C09031=1032.657,-130.353,-79.572,167.440,40.256,157.483
C09032=1032.659,-130.603,-79.558,167.438,40.252,157.482
C09033=1032.660,-130.853,-79.542,167.436,40.248,157.482
C09034=1032.663,-131.102,-79.526,167.435,40.244,157.481
C09035=1032.666,-131.352,-79.509,167.433,40.239,157.480
C09036=1032.671,-131.603,-79.492,167.432,40.234,157.479
C09037=1032.675,-131.852,-79.475,167.431,40.228,157.478
C09038=1032.681,-132.102,-79.456,167.430,40.222,157.477
C09039=1032.354,-132.127,-79.747,167.381,40.451,157.513
C09040=1032.348,-131.877,-79.766,167.383,40.457,157.514
C09041=1032.344,-131.627,-79.784,167.384,40.463,157.515
C09042=1032.340,-131.377,-79.801,167.385,40.468,157.516
C09043=1032.337,-131.127,-79.818,167.386,40.473,157.517
C09044=1032.333,-130.877,-79.834,167.388,40.478,157.518
C09045=1032.331,-130.627,-79.849,167.390,40.482,157.519
C09046=1032.330,-130.377,-79.864,167.391,40.485,157.519
C09047=1032.330,-130.127,-79.879,167.393,40.488,157.520
C09048=1032.330,-129.877,-79.892,167.395,40.490,157.520
C09049=1032.331,-129.628,-79.905,167.397,40.492,157.521
C09050=1032.331,-129.377,-79.918,167.400,40.494,157.521
C09051=1032.334,-129.128,-79.930,167.402,40.495,157.521
C09052=1032.336,-128.878,-79.941,167.404,40.496,157.522
C09053=1032.339,-128.629,-79.952,167.406,40.495,157.522
C09054=1032.343,-128.379,-79.962,167.409,40.495,157.522
C09055=1032.348,-128.129,-79.971,167.411,40.495,157.522
C09056=1032.353,-127.880,-79.981,167.414,40.493,157.522
C09057=1032.359,-127.629,-79.990,167.417,40.492,157.522
C09058=1032.364,-127.380,-79.998,167.419,40.490,157.521
C09059=1032.371,-127.131,-80.007,167.422,40.488,157.521
C09060=1032.376,-126.881,-80.015,167.425,40.487,157.521
C09061=1032.382,-126.631,-80.023,167.428,40.485,157.521
C09062=1032.388,-126.381,-80.032,167.430,40.483,157.521
C09063=1032.395,-126.132,-80.041,167.434,40.482,157.521
C09064=1032.400,-125.882,-80.049,167.437,40.480,157.520
C09065=1032.406,-125.632,-80.058,167.440,40.478,157.520
C09066=1032.412,-125.382,-80.066,167.442,40.477,157.520
C09067=1032.418,-125.132,-80.075,167.445,40.475,157.520
C09068=1032.423,-124.883,-80.084,167.448,40.473,157.520
C09069=1032.430,-124.633,-80.092,167.451,40.472,157.520
C09070=1032.435,-124.383,-80.101,167.453,40.470,157.520
C09071=1032.441,-124.133,-80.110,167.456,40.469,157.520
C09072=1032.447,-123.884,-80.118,167.459,40.467,157.519
C09073=1032.453,-123.633,-80.127,167.462,40.466,157.519
C09074=1032.458,-123.384,-80.136,167.465,40.464,157.519
C09075=1032.465,-123.134,-80.145,167.467,40.462,157.519
C09076=1032.471,-122.884,-80.153,167.470,40.461,157.519
C09077=1032.477,-122.635,-80.163,167.473,40.459,157.519
C09078=1032.482,-122.385,-80.171,167.476,40.457,157.518
C09079=1032.488,-122.134,-80.180,167.479,40.456,157.518
C09080=1032.494,-121.886,-80.189,167.481,40.455,157.518
C09081=1032.500,-121.635,-80.197,167.484,40.453,157.518
C09082=1032.505,-121.386,-80.206,167.487,40.451,157.518
C09083=1032.511,-121.136,-80.216,167.490,40.450,157.518
C09084=1032.517,-120.886,-80.223,167.492,40.448,157.518
C09085=1032.524,-120.637,-80.233,167.496,40.446,157.517
C09086=1032.529,-120.387,-80.241,167.499,40.445,157.517
C09087=1032.535,-120.137,-80.251,167.502,40.444,157.517
C09088=1032.541,-119.887,-80.260,167.504,40.442,157.517
C09089=1032.547,-119.637,-80.268,167.507,40.440,157.517
C09090=1032.553,-119.387,-80.277,167.510,40.439,157.517
C09091=1032.558,-119.138,-80.286,167.513,40.437,157.517
C09092=1032.565,-118.888,-80.295,167.516,40.436,157.517
C09093=1032.570,-118.638,-80.304,167.518,40.435,157.516
C09094=1032.577,-118.389,-80.313,167.521,40.433,157.516
C09095=1032.583,-118.138,-80.322,167.524,40.431,157.516
C09096=1032.588,-117.889,-80.331,167.527,40.430,157.516
C09097=1032.594,-117.639,-80.340,167.529,40.428,157.516
C09098=1032.600,-117.389,-80.349,167.532,40.427,157.516
C09099=1032.606,-117.140,-80.358,167.535,40.425,157.516
C09100=1032.613,-116.853,-80.368,167.538,40.424,157.516
C09101=1032.620,-116.566,-80.379,167.542,40.422,157.515
C09102=1032.626,-116.280,-80.390,167.544,40.420,157.515
C09103=1032.633,-115.994,-80.400,167.548,40.418,157.515
C09104=1032.639,-115.744,-80.409,167.551,40.417,157.515
C09105=1032.645,-115.494,-80.418,167.554,40.415,157.515
C09106=1032.651,-115.245,-80.427,167.556,40.414,157.515
C09107=1032.657,-114.994,-80.436,167.559,40.413,157.515
C09108=1032.663,-114.745,-80.446,167.562,40.411,157.514
C09109=1032.669,-114.495,-80.454,167.565,40.409,157.514
C09110=1032.675,-114.245,-80.463,167.568,40.408,157.514
C09111=1032.681,-113.996,-80.473,167.570,40.407,157.514
C09112=1032.687,-113.747,-80.482,167.573,40.405,157.514
C09113=1032.693,-113.496,-80.491,167.576,40.403,157.514
C09114=1032.699,-113.246,-80.500,167.579,40.402,157.514
C09115=1032.704,-112.997,-80.510,167.582,40.401,157.514
C09116=1032.710,-112.747,-80.518,167.584,40.399,157.513
C09117=1032.716,-112.497,-80.528,167.587,40.398,157.513
C09118=1032.723,-112.247,-80.538,167.590,40.396,157.513
C09119=1032.728,-111.998,-80.547,167.593,40.395,157.513
C09120=1032.734,-111.748,-80.556,167.596,40.394,157.513
C09121=1032.740,-111.498,-80.565,167.598,40.392,157.513
C09122=1032.746,-111.248,-80.575,167.601,40.391,157.513
C09123=1032.752,-110.999,-80.584,167.604,40.390,157.513
C09124=1032.758,-110.749,-80.594,167.607,40.388,157.513
C09125=1032.764,-110.499,-80.602,167.610,40.386,157.512
C09126=1032.770,-110.249,-80.612,167.612,40.385,157.512
C09127=1032.776,-110.000,-80.621,167.615,40.384,157.512
C09128=1032.782,-109.750,-80.631,167.618,40.382,157.512
C09129=1032.787,-109.500,-80.641,167.621,40.381,157.512
C09130=1032.793,-109.250,-80.650,167.624,40.379,157.512
C09131=1032.799,-109.001,-80.660,167.626,40.378,157.512
C09132=1032.805,-108.751,-80.668,167.629,40.377,157.512
C09133=1032.811,-108.501,-80.678,167.632,40.375,157.511
C09134=1032.817,-108.251,-80.688,167.635,40.374,157.511
C09135=1032.823,-108.001,-80.697,167.638,40.373,157.511
C09136=1032.830,-107.751,-80.707,167.640,40.371,157.511
C09137=1032.835,-107.502,-80.716,167.643,40.369,157.511
C09138=1032.841,-107.253,-80.726,167.646,40.368,157.511
C09139=1032.848,-107.003,-80.735,167.649,40.367,157.511
C09140=1032.854,-106.753,-80.745,167.652,40.366,157.511
C09141=1032.860,-106.503,-80.754,167.654,40.364,157.511
C09142=1032.865,-106.253,-80.764,167.656,40.363,157.511
C09143=1032.871,-106.004,-80.774,167.659,40.362,157.510
C09144=1032.877,-105.754,-80.783,167.662,40.361,157.510
C09145=1032.883,-105.504,-80.793,167.665,40.359,157.510
C09146=1032.889,-105.255,-80.802,167.668,40.358,157.510
C09147=1032.895,-105.004,-80.812,167.670,40.356,157.510
C09148=1032.901,-104.755,-80.822,167.673,40.355,157.510
C09149=1032.907,-104.505,-80.832,167.676,40.354,157.510
C09150=1032.913,-104.256,-80.841,167.679,40.352,157.510
C09151=1032.919,-104.006,-80.850,167.682,40.351,157.510
C09152=1032.924,-103.756,-80.861,167.684,40.349,157.509
C09153=1032.931,-103.506,-80.870,167.687,40.349,157.509
C09154=1032.937,-103.256,-80.880,167.690,40.347,157.509
C09155=1032.943,-103.006,-80.889,167.693,40.346,157.509
C09156=1032.949,-102.757,-80.900,167.696,40.344,157.509
C09157=1032.955,-102.507,-80.910,167.699,40.343,157.509
C09158=1032.961,-102.257,-80.919,167.701,40.342,157.509
C09159=1032.967,-102.008,-80.929,167.704,40.341,157.509
C09160=1032.973,-101.758,-80.938,167.707,40.339,157.509
C09161=1032.978,-101.508,-80.948,167.710,40.338,157.509
C09162=1032.984,-101.259,-80.958,167.713,40.337,157.509
C09163=1032.991,-101.009,-80.968,167.715,40.336,157.508
C09164=1032.998,-100.722,-80.979,167.718,40.334,157.508
C09165=1033.004,-100.435,-80.991,167.721,40.333,157.508
C09166=1033.011,-100.148,-81.002,167.725,40.331,157.508
C09167=1033.019,-99.861,-81.013,167.728,40.330,157.508
C09168=1033.024,-99.610,-81.023,167.731,40.329,157.508
C09169=1033.031,-99.361,-81.034,167.733,40.327,157.508
C09170=1033.037,-99.111,-81.043,167.736,40.326,157.508
C09171=1033.043,-98.862,-81.053,167.739,40.324,157.507
C09172=1033.048,-98.612,-81.063,167.742,40.323,157.507
C09173=1033.055,-98.362,-81.073,167.745,40.322,157.507
C09174=1033.061,-98.113,-81.083,167.748,40.321,157.507
C09175=1033.067,-97.863,-81.092,167.750,40.319,157.507
C09176=1033.073,-97.613,-81.103,167.752,40.318,157.507
C09177=1033.079,-97.363,-81.113,167.755,40.317,157.507
C09178=1033.085,-97.113,-81.123,167.758,40.316,157.507
C09179=1033.091,-96.864,-81.133,167.761,40.315,157.507
C09180=1033.096,-96.614,-81.143,167.764,40.314,157.507
C09181=1033.103,-96.364,-81.153,167.767,40.313,157.507
C09182=1033.108,-96.115,-81.164,167.769,40.311,157.507
C09183=1033.115,-95.865,-81.173,167.772,40.310,157.506
C09184=1033.120,-95.615,-81.184,167.775,40.309,157.506
C09185=1033.126,-95.366,-81.194,167.777,40.308,157.506
C09186=1033.132,-95.116,-81.204,167.780,40.307,157.506
C09187=1033.138,-94.866,-81.215,167.783,40.306,157.506
C09188=1033.144,-94.616,-81.224,167.786,40.305,157.506
C09189=1033.150,-94.367,-81.235,167.788,40.303,157.506
C09190=1033.156,-94.117,-81.245,167.791,40.302,157.506
C09191=1033.161,-93.868,-81.256,167.794,40.301,157.506
C09192=1033.168,-93.618,-81.265,167.797,40.300,157.506
C09193=1033.173,-93.368,-81.276,167.800,40.299,157.506
C09194=1033.180,-93.118,-81.286,167.802,40.298,157.506
C09195=1033.186,-92.868,-81.297,167.805,40.297,157.506
C09196=1033.192,-92.618,-81.307,167.808,40.296,157.506
C09197=1033.198,-92.369,-81.317,167.810,40.294,157.505
C09198=1033.204,-92.119,-81.327,167.813,40.293,157.505
C09199=1033.210,-91.870,-81.338,167.816,40.292,157.505
C09200=1033.215,-91.620,-81.348,167.819,40.291,157.505
C09201=1033.222,-91.370,-81.358,167.822,40.290,157.505
C09202=1033.227,-91.121,-81.369,167.824,40.289,157.505
C09203=1033.234,-90.870,-81.379,167.826,40.288,157.505
C09204=1033.240,-90.621,-81.390,167.829,40.286,157.505
C09205=1033.246,-90.371,-81.400,167.832,40.285,157.505
C09206=1033.252,-90.122,-81.410,167.835,40.284,157.505
C09207=1033.257,-89.872,-81.421,167.838,40.283,157.505
C09208=1033.264,-89.622,-81.431,167.841,40.282,157.505
C09209=1033.269,-89.373,-81.442,167.844,40.281,157.504
C09210=1033.276,-89.123,-81.452,167.845,40.280,157.504
C09211=1033.282,-88.873,-81.463,167.848,40.279,157.504
C09212=1033.288,-88.624,-81.473,167.851,40.277,157.504
C09213=1033.294,-88.374,-81.484,167.854,40.276,157.504
C09214=1033.300,-88.124,-81.494,167.857,40.275,157.504
C09215=1033.307,-87.874,-81.505,167.860,40.274,157.504
C09216=1033.312,-87.625,-81.515,167.863,40.274,157.504
C09217=1033.319,-87.375,-81.525,167.865,40.272,157.504
C09218=1033.324,-87.125,-81.536,167.867,40.271,157.504
C09219=1033.331,-86.875,-81.547,167.870,40.270,157.504
C09220=1033.337,-86.626,-81.557,167.873,40.269,157.504
C09221=1033.343,-86.376,-81.568,167.876,40.267,157.504
C09222=1033.349,-86.127,-81.578,167.879,40.267,157.504
C09223=1033.355,-85.877,-81.589,167.882,40.266,157.503
C09224=1033.361,-85.627,-81.600,167.885,40.265,157.503
C09225=1033.367,-85.377,-81.610,167.887,40.263,157.503
C09226=1033.373,-85.128,-81.620,167.889,40.262,157.503
C09227=1033.380,-84.878,-81.631,167.892,40.261,157.503
C09228=1033.387,-84.593,-81.643,167.896,40.260,157.503
C09229=1033.394,-84.309,-81.655,167.899,40.258,157.503
C09230=1033.401,-84.023,-81.667,167.902,40.258,157.503
C09231=1033.408,-83.739,-81.679,167.904,40.256,157.503
C09232=1033.413,-83.489,-81.690,167.907,40.255,157.503
C09233=1033.420,-83.239,-81.701,167.910,40.254,157.503
C09234=1033.426,-82.990,-81.712,167.913,40.253,157.503
C09235=1033.432,-82.740,-81.722,167.916,40.251,157.503
C09236=1033.439,-82.490,-81.733,167.919,40.250,157.502
C09237=1033.444,-82.240,-81.743,167.921,40.250,157.502
C09238=1033.450,-81.991,-81.754,167.924,40.249,157.502
C09239=1033.457,-81.741,-81.765,167.926,40.248,157.502
C09240=1033.463,-81.491,-81.776,167.929,40.246,157.502
C09241=1033.469,-81.242,-81.787,167.932,40.245,157.502
C09242=1033.476,-80.992,-81.797,167.935,40.244,157.502
C09243=1033.481,-80.743,-81.808,167.938,40.243,157.502
C09244=1033.489,-80.493,-81.819,167.940,40.242,157.502
C09245=1033.494,-80.243,-81.830,167.943,40.241,157.502
C09246=1033.500,-79.994,-81.841,167.945,40.240,157.502
C09247=1033.506,-79.744,-81.852,167.948,40.239,157.502
C09248=1033.513,-79.494,-81.862,167.951,40.238,157.502
C09249=1033.519,-79.244,-81.873,167.954,40.237,157.502
C09250=1033.525,-78.995,-81.884,167.956,40.236,157.502
C09251=1033.531,-78.745,-81.895,167.959,40.235,157.502
C09252=1033.537,-78.495,-81.906,167.962,40.234,157.501
C09253=1033.543,-78.245,-81.917,167.965,40.233,157.501
C09254=1033.549,-77.996,-81.928,167.968,40.232,157.501
C09255=1033.555,-77.746,-81.939,167.969,40.231,157.501
C09256=1033.561,-77.496,-81.950,167.972,40.230,157.501
C09257=1033.568,-77.246,-81.961,167.975,40.229,157.501
C09258=1033.574,-76.998,-81.972,167.978,40.228,157.501
///RCONF 1,0,0,1,1,0,0,0,0,0,0,0,0,0,0,0,0,0,0,0,0,0,0,0
C09259=1033.579,-76.748,-81.983,167.981,40.228,157.501
C09260=1033.586,-76.498,-81.995,167.983,40.227,157.501
C09261=1033.592,-76.248,-82.005,167.986,40.226,157.501
C09262=1033.598,-75.998,-82.017,167.989,40.225,157.501
///RCONF 1,0,0,0,1,0,0,0,0,0,0,0,0,0,0,0,0,0,0,0,0,0,0,0
C09263=1033.604,-75.749,-82.028,167.992,40.224,157.501
C09264=1033.610,-75.499,-82.039,167.995,40.223,157.501
C09265=1033.616,-75.250,-82.050,167.996,40.222,157.501
C09266=1033.622,-74.999,-82.062,167.999,40.221,157.501
C09267=1033.628,-74.750,-82.072,168.002,40.219,157.501
C09268=1033.635,-74.500,-82.083,168.005,40.218,157.501
C09269=1033.641,-74.251,-82.094,168.008,40.218,157.501
C09270=1033.647,-74.002,-82.106,168.010,40.217,157.501
C09271=1033.653,-73.751,-82.117,168.013,40.216,157.501
C09272=1033.658,-73.502,-82.128,168.016,40.215,157.500
C09273=1033.665,-73.252,-82.140,168.019,40.214,157.500
///RCONF 1,0,0,0,0,0,0,0,0,0,0,0,0,0,0,0,0,0,0,0,0,0,0,0
C09274=1033.671,-73.003,-82.151,168.020,40.214,157.500
C09275=1033.677,-72.752,-82.162,168.023,40.213,157.500
C09276=1033.683,-72.504,-82.174,168.026,40.212,157.500
C09277=1033.689,-72.253,-82.186,168.028,40.212,157.500
C09278=1033.694,-72.004,-82.197,168.031,40.211,157.500
C09279=1033.701,-71.754,-82.209,168.034,40.210,157.500
C09280=1033.707,-71.505,-82.220,168.037,40.209,157.500
C09281=1033.713,-71.254,-82.231,168.039,40.208,157.500
C09282=1033.718,-71.005,-82.243,168.042,40.208,157.500
C09283=1033.725,-70.755,-82.254,168.045,40.207,157.500
C09284=1033.731,-70.506,-82.266,168.048,40.206,157.500
C09285=1033.737,-70.256,-82.277,168.050,40.205,157.500
C09286=1033.743,-70.006,-82.288,168.052,40.204,157.500
C09287=1033.749,-69.757,-82.300,168.055,40.203,157.500
C09288=1033.755,-69.507,-82.311,168.057,40.203,157.500
C09289=1033.761,-69.257,-82.323,168.060,40.202,157.500
C09290=1033.767,-69.008,-82.334,168.063,40.201,157.500
C09291=1033.774,-68.758,-82.346,168.066,40.200,157.500
C09292=1033.780,-68.476,-82.359,168.069,40.199,157.500
C09293=1033.787,-68.193,-82.372,168.072,40.198,157.500
C09294=1033.794,-67.910,-82.385,168.075,40.197,157.500
C09295=1033.801,-67.628,-82.398,168.078,40.197,157.500
C09296=1033.806,-67.377,-82.410,168.081,40.196,157.500
C09297=1033.813,-67.128,-82.422,168.083,40.195,157.500
C09298=1033.819,-66.878,-82.433,168.085,40.194,157.500
C09299=1033.825,-66.629,-82.445,168.088,40.193,157.500
C09300=1033.831,-66.380,-82.456,168.091,40.192,157.500
C09301=1033.837,-66.129,-82.468,168.093,40.192,157.500
C09302=1033.843,-65.880,-82.480,168.096,40.191,157.500
C09303=1033.849,-65.630,-82.491,168.099,40.190,157.500
C09304=1033.856,-65.381,-82.503,168.101,40.189,157.499
C09305=1033.861,-65.131,-82.514,168.104,40.188,157.499
C09306=1033.868,-64.881,-82.526,168.107,40.188,157.499
C09307=1033.874,-64.632,-82.538,168.110,40.187,157.499
C09308=1033.880,-64.382,-82.549,168.112,40.186,157.499
C09309=1033.886,-64.132,-82.562,168.115,40.185,157.499
C09310=1033.892,-63.882,-82.573,168.117,40.184,157.499
C09311=1033.898,-63.633,-82.585,168.120,40.184,157.499
C09312=1033.905,-63.384,-82.597,168.122,40.183,157.499
C09313=1033.910,-63.133,-82.608,168.125,40.182,157.499
C09314=1033.916,-62.884,-82.620,168.128,40.181,157.499
C09315=1033.923,-62.635,-82.632,168.130,40.180,157.499
C09316=1033.929,-62.384,-82.643,168.133,40.179,157.499
C09317=1033.935,-62.135,-82.656,168.136,40.179,157.499
C09318=1033.941,-61.886,-82.667,168.138,40.178,157.499
C09319=1033.948,-61.636,-82.679,168.141,40.177,157.499
C09320=1033.954,-61.386,-82.691,168.144,40.176,157.499
C09321=1033.960,-61.137,-82.703,168.146,40.175,157.499
C09322=1033.966,-60.887,-82.715,168.149,40.175,157.499
C09323=1033.973,-60.637,-82.726,168.151,40.174,157.499
C09324=1033.979,-60.387,-82.738,168.154,40.173,157.499
C09325=1033.985,-60.138,-82.750,168.156,40.172,157.499
C09326=1033.991,-59.889,-82.762,168.159,40.171,157.499
C09327=1033.998,-59.639,-82.773,168.162,40.171,157.499
C09328=1034.004,-59.389,-82.786,168.164,40.170,157.499
C09329=1034.010,-59.140,-82.797,168.167,40.169,157.499
C09330=1034.016,-58.890,-82.809,168.170,40.168,157.499
C09331=1034.023,-58.640,-82.821,168.172,40.168,157.499
C09332=1034.028,-58.390,-82.833,168.175,40.167,157.499
C09333=1034.035,-58.141,-82.845,168.178,40.166,157.499
C09334=1034.041,-57.892,-82.857,168.180,40.166,157.499
C09335=1034.047,-57.642,-82.869,168.182,40.165,157.499
C09336=1034.054,-57.392,-82.881,168.185,40.164,157.499
C09337=1034.060,-57.142,-82.893,168.188,40.163,157.499
C09338=1034.067,-56.892,-82.905,168.190,40.163,157.499
C09339=1034.073,-56.643,-82.917,168.193,40.162,157.498
C09340=1034.079,-56.394,-82.929,168.196,40.161,157.498
C09341=1034.085,-56.144,-82.941,168.198,40.160,157.498
C09342=1034.091,-55.894,-82.953,168.201,40.159,157.498
C09343=1034.098,-55.645,-82.965,168.204,40.159,157.498
C09344=1034.105,-55.395,-82.977,168.206,40.158,157.498
C09345=1034.110,-55.145,-82.989,168.209,40.157,157.498
C09346=1034.117,-54.895,-83.001,168.212,40.156,157.498
C09347=1034.123,-54.646,-83.012,168.214,40.156,157.498
C09348=1034.129,-54.396,-83.025,168.216,40.155,157.498
C09349=1034.135,-54.147,-83.037,168.219,40.154,157.498
C09350=1034.142,-53.897,-83.049,168.221,40.153,157.498
C09351=1034.148,-53.647,-83.062,168.224,40.152,157.498
C09352=1034.155,-53.398,-83.073,168.227,40.152,157.498
C09353=1034.161,-53.148,-83.085,168.229,40.151,157.498
C09354=1034.167,-52.898,-83.098,168.232,40.150,157.498
C09355=1034.174,-52.649,-83.110,168.235,40.149,157.498
C09356=1034.181,-52.368,-83.124,168.238,40.148,157.498
C09357=1034.188,-52.086,-83.137,168.241,40.147,157.498
C09358=1034.195,-51.805,-83.150,168.244,40.147,157.498
C09359=1034.202,-51.523,-83.165,168.247,40.146,157.498
C09360=1034.209,-51.274,-83.177,168.250,40.145,157.498
C09361=1034.215,-51.024,-83.189,168.251,40.144,157.498
C09362=1034.221,-50.774,-83.201,168.254,40.143,157.498
C09363=1034.228,-50.525,-83.213,168.257,40.143,157.498
C09364=1034.234,-50.275,-83.226,168.259,40.142,157.498
C09365=1034.241,-50.025,-83.238,168.262,40.141,157.498
C09366=1034.247,-49.776,-83.251,168.264,40.141,157.498
C09367=1034.253,-49.526,-83.264,168.267,40.140,157.498
C09368=1034.259,-49.276,-83.276,168.270,40.140,157.498
C09369=1034.265,-49.027,-83.288,168.272,40.139,157.498
C09370=1034.271,-48.778,-83.300,168.275,40.138,157.498
C09371=1034.277,-48.528,-83.314,168.277,40.138,157.498
C09372=1034.283,-48.279,-83.326,168.280,40.137,157.498
C09373=1034.289,-48.029,-83.338,168.282,40.136,157.498
C09374=1034.295,-47.779,-83.351,168.285,40.135,157.498
C09375=1034.302,-47.530,-83.363,168.288,40.135,157.498
C09376=1034.308,-47.280,-83.376,168.290,40.134,157.498
C09377=1034.314,-47.030,-83.388,168.293,40.134,157.498
C09378=1034.320,-46.780,-83.401,168.295,40.133,157.498
C09379=1034.327,-46.531,-83.414,168.298,40.133,157.498
C09380=1034.333,-46.282,-83.426,168.300,40.132,157.498
C09381=1034.339,-46.032,-83.439,168.302,40.132,157.498
C09382=1034.346,-45.783,-83.451,168.305,40.131,157.498
C09383=1034.352,-45.533,-83.464,168.307,40.131,157.498
C09384=1034.357,-45.283,-83.477,168.310,40.130,157.498
C09385=1034.364,-45.034,-83.490,168.313,40.129,157.498
C09386=1034.370,-44.784,-83.502,168.315,40.129,157.498
C09387=1034.376,-44.534,-83.514,168.318,40.128,157.498
C09388=1034.382,-44.285,-83.528,168.320,40.128,157.498
C09389=1034.389,-44.035,-83.540,168.323,40.127,157.498
C09390=1034.395,-43.786,-83.552,168.325,40.126,157.498
C09391=1034.401,-43.536,-83.565,168.328,40.125,157.498
C09392=1034.407,-43.286,-83.578,168.331,40.125,157.498
C09393=1034.414,-43.037,-83.590,168.333,40.124,157.498
C09394=1034.421,-42.787,-83.604,168.336,40.123,157.498
C09395=1034.426,-42.537,-83.616,168.338,40.123,157.498
C09396=1034.433,-42.288,-83.629,168.341,40.122,157.498
C09397=1034.439,-42.038,-83.641,168.343,40.122,157.498
C09398=1034.446,-41.789,-83.655,168.346,40.121,157.498
C09399=1034.451,-41.539,-83.667,168.349,40.121,157.498
C09400=1034.458,-41.290,-83.680,168.350,40.120,157.498
C09401=1034.464,-41.040,-83.692,168.354,40.120,157.498
C09402=1034.470,-40.790,-83.705,168.355,40.119,157.498
C09403=1034.476,-40.541,-83.718,168.358,40.118,157.498
C09404=1034.483,-40.290,-83.731,168.360,40.118,157.498
C09405=1034.490,-40.041,-83.744,168.363,40.117,157.498
C09406=1034.496,-39.792,-83.756,168.366,40.117,157.498
C09407=1034.502,-39.542,-83.770,168.368,40.116,157.498
C09408=1034.508,-39.292,-83.782,168.371,40.115,157.498
C09409=1034.515,-39.043,-83.795,168.373,40.115,157.498
C09410=1034.521,-38.794,-83.808,168.376,40.114,157.498
C09411=1034.528,-38.544,-83.821,168.378,40.113,157.498
C09412=1034.534,-38.294,-83.834,168.381,40.113,157.498
C09413=1034.540,-38.044,-83.847,168.383,40.112,157.498
C09414=1034.546,-37.795,-83.860,168.386,40.112,157.498
C09415=1034.552,-37.546,-83.873,168.388,40.112,157.498
C09416=1034.558,-37.296,-83.886,168.391,40.111,157.498
C09417=1034.564,-37.047,-83.899,168.393,40.111,157.498
C09418=1034.570,-36.798,-83.913,168.396,40.110,157.498
C09419=1034.577,-36.547,-83.925,168.398,40.110,157.498
C09420=1034.583,-36.267,-83.941,168.401,40.109,157.498
C09421=1034.591,-35.985,-83.955,168.404,40.108,157.498
C09422=1034.598,-35.704,-83.970,168.407,40.108,157.498
C09423=1034.604,-35.423,-83.985,168.410,40.107,157.498
C09424=1034.611,-35.174,-83.998,168.412,40.107,157.498
C09425=1034.617,-34.923,-84.011,168.415,40.106,157.498
C09426=1034.623,-34.674,-84.025,168.417,40.106,157.498
C09427=1034.629,-34.425,-84.038,168.420,40.106,157.498
C09428=1034.635,-34.175,-84.050,168.422,40.105,157.498
C09429=1034.642,-33.926,-84.064,168.425,40.104,157.498
C09430=1034.648,-33.676,-84.077,168.426,40.104,157.498
C09431=1034.655,-33.427,-84.091,168.429,40.103,157.498
C09432=1034.661,-33.177,-84.104,168.431,40.103,157.498
C09433=1034.667,-32.927,-84.116,168.434,40.102,157.498
C09434=1034.674,-32.677,-84.130,168.436,40.102,157.498
C09435=1034.680,-32.428,-84.143,168.439,40.101,157.498
C09436=1034.686,-32.179,-84.157,168.441,40.101,157.498
C09437=1034.692,-31.930,-84.170,168.444,40.101,157.498
C09438=1034.699,-31.679,-84.183,168.446,40.100,157.498
C09439=1034.705,-31.430,-84.196,168.449,40.099,157.498
C09440=1034.711,-31.181,-84.209,168.451,40.099,157.498
C09441=1034.717,-30.931,-84.223,168.454,40.098,157.498
C09442=1034.724,-30.681,-84.236,168.456,40.097,157.498
C09443=1034.730,-30.432,-84.249,168.459,40.097,157.498
C09444=1034.737,-30.183,-84.263,168.461,40.097,157.498
C09445=1034.743,-29.932,-84.276,168.464,40.096,157.498
C09446=1034.749,-29.683,-84.289,168.466,40.096,157.498
C09447=1034.756,-29.434,-84.302,168.469,40.095,157.498
C09448=1034.762,-29.184,-84.315,168.471,40.095,157.498
C09449=1034.768,-28.934,-84.330,168.473,40.095,157.498
C09450=1034.774,-28.685,-84.343,168.476,40.094,157.498
C09451=1034.780,-28.436,-84.356,168.478,40.093,157.498
C09452=1034.787,-28.186,-84.370,168.481,40.093,157.498
C09453=1034.793,-27.936,-84.383,168.483,40.092,157.498
C09454=1034.800,-27.686,-84.397,168.486,40.092,157.498
C09455=1034.806,-27.437,-84.410,168.488,40.091,157.498
C09456=1034.813,-27.188,-84.423,168.491,40.091,157.498
C09457=1034.819,-26.938,-84.437,168.493,40.090,157.498
C09458=1034.825,-26.688,-84.451,168.496,40.090,157.498
C09459=1034.831,-26.439,-84.464,168.498,40.090,157.498
C09460=1034.838,-26.189,-84.478,168.501,40.089,157.498
C09461=1034.843,-25.940,-84.492,168.503,40.089,157.498
C09462=1034.850,-25.690,-84.505,168.505,40.088,157.498
C09463=1034.856,-25.440,-84.518,168.508,40.088,157.498
C09464=1034.863,-25.191,-84.532,168.510,40.088,157.498
C09465=1034.868,-24.941,-84.546,168.513,40.087,157.498
C09466=1034.875,-24.692,-84.559,168.515,40.087,157.498
C09467=1034.881,-24.442,-84.572,168.518,40.086,157.498
C09468=1034.887,-24.193,-84.587,168.520,40.086,157.498
C09469=1034.894,-23.943,-84.601,168.522,40.085,157.498
C09470=1034.900,-23.694,-84.614,168.525,40.085,157.498
C09471=1034.906,-23.444,-84.628,168.527,40.085,157.499
C09472=1034.912,-23.195,-84.641,168.530,40.084,157.498
C09473=1034.918,-22.945,-84.655,168.532,40.084,157.499
C09474=1034.924,-22.695,-84.669,168.534,40.084,157.499
C09475=1034.931,-22.446,-84.683,168.537,40.083,157.499
C09476=1034.938,-22.196,-84.697,168.538,40.083,157.499
C09477=1034.943,-21.947,-84.710,168.542,40.082,157.499
C09478=1034.950,-21.697,-84.724,168.544,40.082,157.499
C09479=1034.956,-21.448,-84.737,168.547,40.082,157.499
C09480=1034.962,-21.199,-84.752,168.548,40.081,157.499
C09481=1034.969,-20.949,-84.766,168.550,40.081,157.499
C09482=1034.975,-20.699,-84.779,168.554,40.081,157.499
C09483=1034.981,-20.449,-84.793,168.555,40.080,157.499
C09484=1034.988,-20.168,-84.809,168.558,40.079,157.499
C09485=1034.995,-19.886,-84.824,168.561,40.079,157.499
C09486=1035.002,-19.604,-84.840,168.563,40.079,157.499
C09487=1035.010,-19.323,-84.856,168.566,40.078,157.499
C09488=1035.016,-19.073,-84.869,168.568,40.078,157.499
C09489=1035.023,-18.823,-84.883,168.571,40.078,157.499
C09490=1035.029,-18.574,-84.898,168.573,40.077,157.499
C09491=1035.035,-18.324,-84.911,168.576,40.076,157.499
C09492=1035.042,-18.075,-84.924,168.578,40.076,157.499
C09493=1035.048,-17.825,-84.939,168.581,40.076,157.499
C09494=1035.054,-17.576,-84.953,168.583,40.075,157.499
C09495=1035.060,-17.326,-84.967,168.585,40.075,157.499
C09496=1035.067,-17.076,-84.981,168.588,40.075,157.499
C09497=1035.074,-16.827,-84.995,168.590,40.074,157.499
C09498=1035.080,-16.577,-85.009,168.593,40.074,157.499
C09499=1035.086,-16.328,-85.023,168.595,40.073,157.499
C09500=1035.093,-16.079,-85.036,168.597,40.073,157.499
C09501=1035.099,-15.829,-85.050,168.600,40.072,157.499
C09502=1035.106,-15.580,-85.065,168.602,40.072,157.499
C09503=1035.111,-15.330,-85.078,168.604,40.072,157.499
C09504=1035.118,-15.081,-85.093,168.607,40.072,157.499
C09505=1035.124,-14.831,-85.107,168.609,40.071,157.499
C09506=1035.131,-14.582,-85.121,168.612,40.070,157.499
C09507=1035.136,-14.332,-85.135,168.614,40.070,157.499
C09508=1035.143,-14.083,-85.150,168.616,40.070,157.499
C09509=1035.150,-13.833,-85.163,168.619,40.070,157.500
C09510=1035.155,-13.584,-85.178,168.621,40.070,157.500
C09511=1035.161,-13.333,-85.192,168.623,40.069,157.500
C09512=1035.168,-13.085,-85.206,168.626,40.069,157.500
C09513=1035.174,-12.834,-85.220,168.628,40.068,157.500
C09514=1035.181,-12.586,-85.234,168.630,40.068,157.500
C09515=1035.187,-12.335,-85.249,168.633,40.068,157.500
C09516=1035.193,-12.086,-85.264,168.635,40.068,157.500
C09517=1035.199,-11.837,-85.277,168.637,40.068,157.500
C09518=1035.206,-11.587,-85.292,168.640,40.067,157.500
C09519=1035.211,-11.338,-85.306,168.642,40.066,157.500
C09520=1035.218,-11.088,-85.320,168.644,40.066,157.500
C09521=1035.224,-10.839,-85.335,168.647,40.066,157.500
C09522=1035.230,-10.589,-85.349,168.649,40.066,157.500
C09523=1035.237,-10.339,-85.363,168.651,40.066,157.500
C09524=1035.243,-10.090,-85.378,168.654,40.065,157.500
C09525=1035.250,-9.840,-85.391,168.656,40.064,157.500
C09526=1035.256,-9.591,-85.406,168.658,40.064,157.500
C09527=1035.262,-9.342,-85.421,168.661,40.064,157.500
C09528=1035.269,-9.092,-85.435,168.663,40.064,157.500
C09529=1035.275,-8.842,-85.450,168.665,40.064,157.500
C09530=1035.281,-8.593,-85.464,168.668,40.063,157.500
C09531=1035.288,-8.343,-85.478,168.670,40.062,157.500
C09532=1035.294,-8.094,-85.493,168.672,40.062,157.500
C09533=1035.300,-7.845,-85.507,168.675,40.062,157.500
C09534=1035.307,-7.595,-85.521,168.677,40.062,157.500
C09535=1035.313,-7.345,-85.536,168.679,40.062,157.500
C09536=1035.319,-7.096,-85.550,168.682,40.061,157.501
C09537=1035.326,-6.847,-85.565,168.684,40.061,157.500
C09538=1035.332,-6.596,-85.579,168.686,40.060,157.501
C09539=1035.338,-6.348,-85.594,168.689,40.060,157.501
C09540=1035.345,-6.098,-85.608,168.691,40.060,157.501
C09541=1035.351,-5.849,-85.623,168.693,40.060,157.501
C09542=1035.357,-5.599,-85.637,168.696,40.059,157.501
C09543=1035.364,-5.350,-85.651,168.698,40.059,157.501
C09544=1035.370,-5.100,-85.666,168.700,40.058,157.501
C09545=1035.377,-4.850,-85.681,168.703,40.058,157.501
C09546=1035.383,-4.601,-85.694,168.705,40.058,157.501
C09547=1035.389,-4.351,-85.709,168.707,40.058,157.501
C09548=1035.396,-4.068,-85.726,168.710,40.057,157.501
C09549=1035.404,-3.785,-85.743,168.712,40.057,157.501
C09550=1035.411,-3.502,-85.759,168.715,40.056,157.501
C09551=1035.419,-3.217,-85.776,168.718,40.056,157.501
C09552=1035.424,-2.968,-85.790,168.720,40.056,157.501
C09553=1035.431,-2.719,-85.805,168.722,40.056,157.501
C09554=1035.437,-2.469,-85.820,168.724,40.056,157.501
C09555=1035.443,-2.220,-85.835,168.727,40.055,157.501
C09556=1035.449,-1.971,-85.850,168.730,40.055,157.501
C09557=1035.456,-1.721,-85.865,168.732,40.055,157.501
C09558=1035.462,-1.471,-85.880,168.734,40.055,157.501
C09559=1035.468,-1.222,-85.894,168.737,40.054,157.501
C09560=1035.474,-0.973,-85.909,168.739,40.054,157.502
C09561=1035.481,-0.723,-85.924,168.741,40.054,157.502
C09562=1035.487,-0.473,-85.939,168.743,40.054,157.502
C09563=1035.493,-0.224,-85.954,168.746,40.054,157.502
C09564=1035.499,0.025,-85.969,168.748,40.053,157.502
C09565=1035.505,0.275,-85.984,168.750,40.053,157.502
C09566=1035.512,0.525,-85.998,168.752,40.053,157.502
C09567=1035.518,0.774,-86.013,168.755,40.053,157.502
C09568=1035.524,1.023,-86.028,168.757,40.053,157.502
C09569=1035.530,1.273,-86.043,168.759,40.052,157.502
C09570=1035.537,1.523,-86.058,168.761,40.052,157.502
C09571=1035.543,1.772,-86.072,168.764,40.052,157.502
C09572=1035.549,2.021,-86.087,168.766,40.052,157.502
C09573=1035.555,2.271,-86.102,168.768,40.052,157.502
C09574=1035.562,2.520,-86.117,168.770,40.051,157.502
C09575=1035.568,2.770,-86.134,168.773,40.051,157.502
C09576=1035.574,3.020,-86.148,168.775,40.051,157.502
C09577=1035.580,3.268,-86.163,168.777,40.051,157.502
C09578=1035.586,3.518,-86.178,168.779,40.051,157.502
C09579=1035.593,3.768,-86.193,168.782,40.050,157.503
C09580=1035.599,4.017,-86.208,168.784,40.050,157.503
C09581=1035.605,4.267,-86.223,168.786,40.050,157.503
C09582=1035.612,4.516,-86.239,168.788,40.050,157.503
C09583=1035.618,4.765,-86.253,168.791,40.049,157.503
C09584=1035.624,5.015,-86.268,168.793,40.049,157.503
C09585=1035.631,5.264,-86.283,168.795,40.049,157.503
C09586=1035.637,5.514,-86.298,168.797,40.049,157.503
C09587=1035.643,5.764,-86.313,168.800,40.049,157.503
C09588=1035.650,6.013,-86.329,168.802,40.048,157.503
C09589=1035.656,6.262,-86.343,168.804,40.048,157.503
C09590=1035.663,6.512,-86.358,168.806,40.048,157.503
C09591=1035.669,6.761,-86.373,168.808,40.048,157.503
C09592=1035.675,7.011,-86.388,168.811,40.048,157.503
C09593=1035.682,7.260,-86.404,168.813,40.047,157.503
C09594=1035.688,7.509,-86.419,168.815,40.047,157.503
C09595=1035.694,7.759,-86.434,168.817,40.047,157.503
C09596=1035.701,8.009,-86.448,168.820,40.046,157.503
C09597=1035.707,8.258,-86.465,168.822,40.046,157.503
C09598=1035.713,8.508,-86.480,168.824,40.046,157.503
C09599=1035.720,8.757,-86.495,168.826,40.046,157.503
C09600=1035.726,9.006,-86.510,168.829,40.045,157.504
C09601=1035.733,9.256,-86.525,168.831,40.045,157.504
C09602=1035.739,9.506,-86.540,168.834,40.045,157.504
C09603=1035.745,9.755,-86.555,168.836,40.045,157.504
C09604=1035.752,10.004,-86.571,168.839,40.045,157.504
C09605=1035.758,10.254,-86.586,168.841,40.044,157.504
C09606=1035.765,10.504,-86.601,168.843,40.044,157.504
C09607=1035.772,10.753,-86.616,168.845,40.044,157.504
C09608=1035.777,11.002,-86.631,168.847,40.044,157.504
C09609=1035.784,11.251,-86.646,168.850,40.043,157.504
C09610=1035.790,11.500,-86.662,168.852,40.043,157.504
C09611=1035.796,11.750,-86.677,168.854,40.043,157.504
C09612=1035.804,12.036,-86.695,168.857,40.042,157.504
C09613=1035.811,12.321,-86.712,168.859,40.042,157.504
C09614=1035.818,12.607,-86.729,168.862,40.042,157.504
C09615=1035.826,12.892,-86.747,168.864,40.042,157.504
C09616=1035.833,13.141,-86.763,168.867,40.041,157.504
C09617=1035.839,13.391,-86.778,168.869,40.041,157.504
C09618=1035.845,13.640,-86.793,168.871,40.041,157.504
C09619=1035.852,13.889,-86.808,168.873,40.041,157.504
C09620=1035.858,14.139,-86.823,168.875,40.041,157.504
C09621=1035.864,14.388,-86.839,168.878,40.040,157.505
C09622=1035.871,14.638,-86.854,168.880,40.040,157.505
C09623=1035.877,14.887,-86.870,168.882,40.040,157.505
C09624=1035.883,15.137,-86.886,168.884,40.040,157.505
C09625=1035.890,15.386,-86.901,168.886,40.040,157.505
C09626=1035.896,15.636,-86.916,168.888,40.039,157.505
C09627=1035.902,15.885,-86.932,168.891,40.039,157.505
C09628=1035.909,16.134,-86.948,168.893,40.039,157.505
C09629=1035.914,16.384,-86.964,168.895,40.039,157.505
C09630=1035.921,16.633,-86.979,168.897,40.039,157.505
C09631=1035.928,16.883,-86.994,168.899,40.039,157.505
C09632=1035.934,17.133,-87.011,168.902,40.039,157.505
C09633=1035.941,17.382,-87.027,168.904,40.039,157.505
C09634=1035.947,17.631,-87.042,168.906,40.038,157.505
C09635=1035.953,17.881,-87.058,168.908,40.038,157.505
C09636=1035.959,18.130,-87.073,168.910,40.038,157.505
C09637=1035.966,18.379,-87.088,168.912,40.038,157.505
C09638=1035.972,18.629,-87.105,168.915,40.038,157.506
C09639=1035.978,18.878,-87.120,168.917,40.037,157.506
C09640=1035.985,19.127,-87.135,168.919,40.037,157.506
C09641=1035.991,19.377,-87.152,168.921,40.037,157.506
C09642=1035.998,19.626,-87.166,168.923,40.037,157.506
C09643=1036.003,19.876,-87.183,168.925,40.037,157.506
C09644=1036.010,20.125,-87.198,168.929,40.036,157.506
C09645=1036.016,20.376,-87.214,168.931,40.036,157.506
C09646=1036.023,20.625,-87.230,168.933,40.037,157.506
C09647=1036.029,20.874,-87.246,168.935,40.036,157.506
C09648=1036.036,21.123,-87.262,168.937,40.036,157.506
C09649=1036.041,21.373,-87.277,168.939,40.036,157.506
C09650=1036.048,21.622,-87.293,168.941,40.036,157.506
C09651=1036.054,21.871,-87.309,168.944,40.036,157.506
C09652=1036.061,22.120,-87.325,168.946,40.035,157.506
C09653=1036.066,22.370,-87.341,168.948,40.035,157.506
C09654=1036.074,22.620,-87.357,168.950,40.035,157.506
C09655=1036.080,22.869,-87.373,168.952,40.035,157.507
C09656=1036.086,23.118,-87.388,168.954,40.035,157.507
C09657=1036.092,23.368,-87.405,168.956,40.035,157.507
C09658=1036.099,23.617,-87.420,168.959,40.035,157.507
C09659=1036.105,23.867,-87.436,168.961,40.035,157.507
C09660=1036.111,24.116,-87.452,168.963,40.034,157.507
C09661=1036.118,24.366,-87.468,168.965,40.034,157.507
C09662=1036.125,24.615,-87.484,168.967,40.034,157.507
C09663=1036.130,24.864,-87.500,168.969,40.034,157.507
C09664=1036.137,25.113,-87.516,168.971,40.034,157.507
C09665=1036.143,25.363,-87.531,168.974,40.033,157.507
C09666=1036.149,25.612,-87.547,168.976,40.033,157.507
C09667=1036.156,25.862,-87.564,168.978,40.033,157.507
C09668=1036.163,26.111,-87.579,168.980,40.034,157.507
C09669=1036.169,26.361,-87.596,168.983,40.033,157.507
C09670=1036.175,26.610,-87.612,168.985,40.033,157.508
C09671=1036.181,26.859,-87.627,168.987,40.033,157.508
C09672=1036.188,27.109,-87.644,168.990,40.033,157.508
C09673=1036.195,27.358,-87.660,168.992,40.033,157.508
C09674=1036.201,27.608,-87.676,168.994,40.032,157.508
C09675=1036.206,27.857,-87.692,168.996,40.032,157.508
C09676=1036.214,28.144,-87.710,168.998,40.032,157.508
C09677=1036.221,28.430,-87.729,169.001,40.032,157.508
C09678=1036.229,28.717,-87.748,169.003,40.032,157.508
C09679=1036.236,29.004,-87.766,169.006,40.032,157.508
C09680=1036.242,29.253,-87.782,169.008,40.032,157.508
C09681=1036.248,29.503,-87.798,169.010,40.032,157.508
C09682=1036.255,29.752,-87.814,169.012,40.031,157.508
C09683=1036.261,30.002,-87.831,169.014,40.032,157.508
C09684=1036.267,30.250,-87.848,169.016,40.032,157.509
C09685=1036.273,30.500,-87.864,169.018,40.031,157.509
C09686=1036.280,30.749,-87.879,169.020,40.031,157.509
C09687=1036.286,30.998,-87.896,169.022,40.031,157.509
C09688=1036.293,31.248,-87.912,169.025,40.031,157.509
C09689=1036.299,31.497,-87.929,169.027,40.031,157.509
C09690=1036.304,31.747,-87.945,169.029,40.031,157.509
C09691=1036.311,31.996,-87.961,169.031,40.031,157.509
C09692=1036.318,32.246,-87.977,169.033,40.031,157.509
C09693=1036.324,32.495,-87.993,169.035,40.031,157.509
C09694=1036.330,32.744,-88.010,169.037,40.030,157.509
C09695=1036.337,32.994,-88.026,169.040,40.031,157.509
C09696=1036.343,33.243,-88.043,169.042,40.031,157.509
C09697=1036.349,33.492,-88.059,169.045,40.030,157.509
C09698=1036.355,33.742,-88.075,169.047,40.030,157.509
C09699=1036.362,33.992,-88.091,169.049,40.030,157.510
C09700=1036.369,34.240,-88.108,169.051,40.030,157.510
C09701=1036.375,34.490,-88.124,169.053,40.030,157.510
C09702=1036.381,34.740,-88.141,169.055,40.030,157.510
C09703=1036.387,34.989,-88.157,169.057,40.030,157.510
C09704=1036.394,35.238,-88.173,169.059,40.030,157.510
C09705=1036.401,35.487,-88.190,169.061,40.030,157.510
C09706=1036.407,35.737,-88.207,169.063,40.029,157.510
C09707=1036.413,35.986,-88.223,169.066,40.029,157.510
C09708=1036.419,36.236,-88.239,169.068,40.029,157.510
C09709=1036.426,36.485,-88.256,169.070,40.029,157.510
C09710=1036.432,36.734,-88.272,169.072,40.029,157.510
C09711=1036.439,36.984,-88.289,169.074,40.029,157.510
C09712=1036.445,37.233,-88.305,169.076,40.029,157.510
C09713=1036.451,37.482,-88.322,169.078,40.029,157.510
C09714=1036.457,37.732,-88.339,169.080,40.028,157.510
C09715=1036.463,37.982,-88.355,169.083,40.029,157.511
C09716=1036.470,38.230,-88.372,169.085,40.029,157.511
C09717=1036.476,38.480,-88.388,169.087,40.029,157.511
C09718=1036.482,38.730,-88.405,169.089,40.028,157.511
C09719=1036.488,38.978,-88.422,169.092,40.029,157.511
C09720=1036.495,39.228,-88.438,169.094,40.029,157.511
C09721=1036.501,39.478,-88.454,169.096,40.028,157.511
C09722=1036.508,39.727,-88.472,169.098,40.028,157.511
C09723=1036.514,39.977,-88.488,169.100,40.029,157.511
C09724=1036.520,40.225,-88.505,169.102,40.028,157.511
C09725=1036.526,40.475,-88.522,169.104,40.028,157.511
C09726=1036.532,40.725,-88.538,169.106,40.028,157.511
C09727=1036.539,40.973,-88.555,169.108,40.028,157.511
C09728=1036.545,41.223,-88.572,169.110,40.028,157.512
C09729=1036.551,41.472,-88.589,169.112,40.028,157.512
C09730=1036.558,41.722,-88.605,169.114,40.028,157.512
C09731=1036.564,41.971,-88.622,169.116,40.028,157.512
C09732=1036.570,42.220,-88.638,169.118,40.028,157.512
C09733=1036.577,42.470,-88.656,169.120,40.028,157.512
C09734=1036.583,42.719,-88.672,169.124,40.028,157.512
C09735=1036.590,42.969,-88.689,169.126,40.028,157.512
C09736=1036.596,43.218,-88.706,169.128,40.027,157.512
C09737=1036.602,43.467,-88.723,169.130,40.028,157.512
C09738=1036.608,43.717,-88.740,169.132,40.028,157.512
C09739=1036.614,43.966,-88.757,169.134,40.028,157.512
C09740=1036.621,44.253,-88.776,169.136,40.028,157.513
C09741=1036.628,44.540,-88.796,169.138,40.028,157.513
C09742=1036.635,44.825,-88.815,169.141,40.028,157.513
C09743=1036.643,45.112,-88.835,169.143,40.028,157.513
C09744=1036.652,45.527,-88.863,169.146,40.028,157.513
C09745=1036.663,45.942,-88.891,169.150,40.028,157.513
C09746=1036.674,46.356,-88.920,169.154,40.028,157.513
C09747=1036.684,46.771,-88.948,169.158,40.028,157.513
C09748=1036.690,47.022,-88.965,169.160,40.029,157.514
C09749=1036.696,47.270,-88.982,169.162,40.028,157.514
C09750=1036.702,47.519,-88.999,169.164,40.028,157.514
C09751=1036.708,47.769,-89.017,169.166,40.029,157.514
C09752=1036.714,48.018,-89.033,169.168,40.028,157.514
C09753=1036.721,48.268,-89.051,169.170,40.028,157.514
C09754=1036.727,48.517,-89.068,169.172,40.029,157.514
C09755=1036.733,48.767,-89.085,169.174,40.029,157.514
C09756=1036.740,49.015,-89.102,169.176,40.028,157.514
C09757=1036.747,49.265,-89.119,169.178,40.028,157.514
C09758=1036.752,49.515,-89.136,169.180,40.029,157.515
C09759=1036.759,49.764,-89.154,169.182,40.028,157.515
C09760=1036.765,50.013,-89.170,169.184,40.028,157.515
C09761=1036.771,50.262,-89.188,169.187,40.029,157.515
C09762=1036.777,50.512,-89.205,169.189,40.029,157.515
C09763=1036.784,50.761,-89.222,169.191,40.028,157.515
C09764=1036.789,51.010,-89.240,169.193,40.029,157.515
C09765=1036.796,51.260,-89.257,169.195,40.029,157.515
C09766=1036.802,51.508,-89.274,169.197,40.028,157.515
C09767=1036.808,51.759,-89.291,169.199,40.028,157.515
C09768=1036.815,52.008,-89.308,169.201,40.029,157.515
C09769=1036.821,52.257,-89.325,169.203,40.029,157.515
C09770=1036.827,52.507,-89.343,169.205,40.028,157.515
C09771=1036.834,52.755,-89.360,169.207,40.029,157.516
C09772=1036.840,53.005,-89.377,169.209,40.029,157.516
C09773=1036.846,53.254,-89.395,169.211,40.028,157.516
C09774=1036.853,53.504,-89.412,169.213,40.028,157.516
C09775=1036.859,53.753,-89.429,169.215,40.029,157.516
C09776=1036.865,54.002,-89.447,169.217,40.029,157.516
C09777=1036.871,54.251,-89.464,169.219,40.028,157.516
C09778=1036.878,54.501,-89.481,169.222,40.028,157.516
C09779=1036.884,54.750,-89.499,169.225,40.029,157.516
C09780=1036.890,55.000,-89.515,169.227,40.028,157.516
C09781=1036.897,55.249,-89.533,169.229,40.028,157.516
C09782=1036.903,55.498,-89.550,169.231,40.029,157.517
C09783=1036.909,55.748,-89.567,169.233,40.028,157.517
C09784=1036.916,55.997,-89.585,169.235,40.028,157.517
C09785=1036.922,56.246,-89.602,169.237,40.028,157.517
C09786=1036.929,56.495,-89.620,169.239,40.029,157.517
C09787=1036.936,56.745,-89.637,169.241,40.028,157.517
C09788=1036.941,56.994,-89.655,169.243,40.028,157.517
C09789=1036.948,57.243,-89.672,169.245,40.028,157.517
C09790=1036.954,57.492,-89.689,169.247,40.028,157.517
C09791=1036.960,57.742,-89.707,169.249,40.028,157.517
C09792=1036.967,57.991,-89.724,169.251,40.028,157.517
C09793=1036.973,58.240,-89.742,169.253,40.028,157.517
C09794=1036.980,58.490,-89.759,169.255,40.028,157.517
C09795=1036.986,58.739,-89.776,169.258,40.028,157.518
C09796=1036.992,58.988,-89.794,169.260,40.028,157.518
C09797=1036.999,59.238,-89.811,169.262,40.028,157.518
C09798=1037.006,59.487,-89.829,169.264,40.028,157.518
C09799=1037.011,59.736,-89.846,169.266,40.028,157.518
C09800=1037.021,60.107,-89.872,169.269,40.028,157.518
C09801=1037.030,60.476,-89.897,169.273,40.027,157.518
C09802=1037.040,60.846,-89.924,169.276,40.027,157.518
C09803=1037.050,61.217,-89.950,169.279,40.028,157.518
C09804=1037.056,61.466,-89.967,169.281,40.027,157.518
C09805=1037.063,61.715,-89.985,169.283,40.027,157.518
C09806=1037.069,61.965,-90.002,169.285,40.027,157.518
C09807=1037.075,62.213,-90.020,169.287,40.027,157.519
C09808=1037.082,62.462,-90.037,169.289,40.027,157.519
C09809=1037.088,62.712,-90.055,169.291,40.027,157.519
C09810=1037.095,62.961,-90.073,169.293,40.027,157.519
C09811=1037.101,63.210,-90.090,169.295,40.027,157.519
C09812=1037.108,63.460,-90.108,169.297,40.026,157.519
C09813=1037.114,63.709,-90.125,169.300,40.027,157.519
C09814=1037.121,63.958,-90.144,169.302,40.027,157.519
C09815=1037.126,64.207,-90.161,169.304,40.027,157.519
C09816=1037.133,64.457,-90.179,169.306,40.027,157.519
C09817=1037.139,64.707,-90.196,169.308,40.027,157.519
C09818=1037.145,64.956,-90.214,169.310,40.027,157.519
C09819=1037.152,65.205,-90.232,169.312,40.027,157.519
C09820=1037.158,65.454,-90.250,169.314,40.027,157.520
C09821=1037.164,65.704,-90.268,169.316,40.027,157.520
C09822=1037.171,65.953,-90.285,169.318,40.027,157.520
C09823=1037.177,66.202,-90.304,169.320,40.027,157.520
C09824=1037.183,66.452,-90.322,169.322,40.027,157.520
C09825=1037.190,66.701,-90.339,169.324,40.027,157.520
C09826=1037.196,66.950,-90.357,169.326,40.027,157.520
C09827=1037.202,67.199,-90.375,169.328,40.027,157.520
C09828=1037.209,67.449,-90.392,169.331,40.027,157.520
C09829=1037.215,67.698,-90.411,169.333,40.027,157.520
C09830=1037.221,67.947,-90.429,169.335,40.027,157.520
C09831=1037.227,68.197,-90.447,169.337,40.027,157.521
C09832=1037.234,68.445,-90.465,169.339,40.027,157.521
C09833=1037.240,68.695,-90.483,169.341,40.027,157.521
C09834=1037.246,68.945,-90.500,169.343,40.028,157.521
C09835=1037.252,69.193,-90.519,169.345,40.027,157.521
C09836=1037.259,69.443,-90.536,169.347,40.027,157.521
C09837=1037.265,69.692,-90.555,169.349,40.028,157.521
C09838=1037.271,69.942,-90.573,169.351,40.027,157.521
C09839=1037.278,70.191,-90.591,169.353,40.028,157.521
C09840=1037.283,70.440,-90.609,169.355,40.028,157.521
C09841=1037.289,70.689,-90.627,169.357,40.028,157.521
C09842=1037.297,70.938,-90.645,169.360,40.028,157.522
C09843=1037.303,71.188,-90.663,169.362,40.028,157.522
C09844=1037.309,71.437,-90.681,169.364,40.028,157.522
C09845=1037.315,71.686,-90.699,169.366,40.028,157.522
C09846=1037.321,71.935,-90.718,169.368,40.028,157.522
C09847=1037.327,72.185,-90.736,169.370,40.028,157.522
C09848=1037.334,72.434,-90.754,169.372,40.028,157.522
C09849=1037.341,72.684,-90.772,169.374,40.029,157.522
C09850=1037.346,72.932,-90.790,169.376,40.028,157.522
C09851=1037.352,73.182,-90.808,169.378,40.028,157.522
C09852=1037.359,73.431,-90.826,169.380,40.029,157.523
C09853=1037.365,73.681,-90.844,169.382,40.029,157.523
C09854=1037.371,73.930,-90.863,169.384,40.028,157.523
C09855=1037.378,74.179,-90.882,169.386,40.029,157.523
C09856=1037.383,74.428,-90.899,169.388,40.029,157.523
C09857=1037.390,74.677,-90.918,169.391,40.029,157.523
C09858=1037.396,74.927,-90.936,169.393,40.029,157.523
C09859=1037.403,75.176,-90.954,169.395,40.029,157.523
C09860=1037.409,75.425,-90.972,169.397,40.029,157.523
C09861=1037.416,75.674,-90.990,169.399,40.029,157.523
C09862=1037.422,75.924,-91.009,169.402,40.029,157.523
C09863=1037.428,76.173,-91.027,169.404,40.029,157.524
C09864=1037.435,76.459,-91.048,169.406,40.029,157.524
C09865=1037.443,76.745,-91.069,169.408,40.029,157.524
C09866=1037.450,77.030,-91.090,169.410,40.029,157.524
C09867=1037.457,77.317,-91.111,169.413,40.030,157.524
C09868=1037.463,77.566,-91.130,169.415,40.029,157.524
C09869=1037.470,77.815,-91.148,169.417,40.029,157.524
C09870=1037.476,78.065,-91.167,169.420,40.030,157.524
C09871=1037.482,78.314,-91.185,169.422,40.030,157.524
C09872=1037.488,78.563,-91.203,169.424,40.030,157.525
C09873=1037.494,78.812,-91.222,169.426,40.030,157.525
C09874=1037.500,79.061,-91.241,169.428,40.030,157.525
C09875=1037.506,79.311,-91.259,169.430,40.030,157.525
C09876=1037.513,79.560,-91.278,169.432,40.031,157.525
C09877=1037.519,79.809,-91.296,169.434,40.030,157.525
C09878=1037.525,80.058,-91.315,169.436,40.031,157.525
C09879=1037.532,80.308,-91.333,169.438,40.031,157.525
C09880=1037.537,80.558,-91.352,169.441,40.031,157.525
C09881=1037.543,80.806,-91.370,169.443,40.031,157.525
C09882=1037.549,81.055,-91.389,169.445,40.031,157.525
C09883=1037.556,81.304,-91.408,169.447,40.031,157.526
C09884=1037.562,81.553,-91.426,169.449,40.031,157.526
C09885=1037.568,81.803,-91.444,169.451,40.031,157.526
C09886=1037.574,82.052,-91.463,169.453,40.031,157.526
C09887=1037.581,82.302,-91.482,169.454,40.032,157.526
C09888=1037.587,82.551,-91.501,169.456,40.032,157.526
C09889=1037.593,82.800,-91.519,169.458,40.032,157.526
C09890=1037.600,83.049,-91.538,169.460,40.032,157.526
C09891=1037.606,83.298,-91.557,169.462,40.032,157.527
C09892=1037.612,83.548,-91.576,169.464,40.032,157.527
C09893=1037.618,83.797,-91.594,169.467,40.033,157.527
C09894=1037.624,84.046,-91.613,169.469,40.032,157.527
C09895=1037.631,84.296,-91.631,169.471,40.032,157.527
C09896=1037.637,84.545,-91.650,169.473,40.033,157.527
C09897=1037.643,84.794,-91.669,169.475,40.033,157.527
C09898=1037.649,85.043,-91.688,169.477,40.033,157.527
C09899=1037.656,85.292,-91.706,169.479,40.033,157.527
C09900=1037.662,85.541,-91.725,169.482,40.033,157.527
C09901=1037.669,85.791,-91.744,169.484,40.033,157.527
C09902=1037.674,86.040,-91.763,169.486,40.033,157.528
C09903=1037.681,86.289,-91.782,169.488,40.033,157.528
C09904=1037.687,86.538,-91.800,169.490,40.033,157.528
C09905=1037.694,86.787,-91.819,169.493,40.034,157.528
C09906=1037.700,87.036,-91.837,169.495,40.033,157.528
C09907=1037.706,87.286,-91.857,169.497,40.034,157.528
C09908=1037.712,87.535,-91.875,169.499,40.034,157.528
C09909=1037.719,87.784,-91.894,169.501,40.033,157.528
C09910=1037.725,88.033,-91.913,169.503,40.034,157.528
C09911=1037.732,88.282,-91.931,169.505,40.034,157.528
C09912=1037.737,88.532,-91.951,169.507,40.034,157.529
C09913=1037.744,88.781,-91.969,169.509,40.034,157.529
C09914=1037.750,89.030,-91.988,169.511,40.034,157.529
C09915=1037.756,89.279,-92.007,169.513,40.034,157.529
C09916=1037.762,89.529,-92.026,169.515,40.034,157.529
C09917=1037.769,89.778,-92.045,169.518,40.035,157.529
C09918=1037.776,90.028,-92.063,169.520,40.034,157.529
C09919=1037.782,90.277,-92.082,169.522,40.035,157.529
C09920=1037.788,90.526,-92.101,169.524,40.035,157.529
C09921=1037.794,90.775,-92.121,169.526,40.035,157.530
C09922=1037.800,91.024,-92.140,169.528,40.035,157.530
C09923=1037.807,91.273,-92.159,169.530,40.035,157.530
C09924=1037.812,91.523,-92.178,169.532,40.035,157.530
C09925=1037.819,91.772,-92.196,169.534,40.036,157.530
C09926=1037.825,92.021,-92.216,169.536,40.035,157.530
C09927=1037.831,92.270,-92.235,169.538,40.036,157.530
C09928=1037.838,92.556,-92.257,169.540,40.036,157.530
C09929=1037.845,92.842,-92.280,169.543,40.036,157.530
C09930=1037.852,93.128,-92.301,169.546,40.037,157.531
C09931=1037.859,93.413,-92.323,169.548,40.036,157.531
C09932=1037.866,93.663,-92.342,169.550,40.037,157.531
C09933=1037.872,93.913,-92.361,169.552,40.037,157.531
C09934=1037.878,94.162,-92.380,169.554,40.037,157.531
C09935=1037.884,94.411,-92.400,169.556,40.037,157.531
C09936=1037.890,94.660,-92.419,169.558,40.037,157.531
C09937=1037.896,94.909,-92.438,169.560,40.037,157.531
C09938=1037.903,95.158,-92.457,169.563,40.038,157.532
C09939=1037.909,95.407,-92.477,169.565,40.037,157.532
C09940=1037.915,95.656,-92.495,169.567,40.038,157.532
C09941=1037.922,95.906,-92.516,169.569,40.038,157.532
C09942=1037.928,96.155,-92.534,169.571,40.038,157.532
C09943=1037.934,96.404,-92.553,169.573,40.038,157.532
C09944=1037.940,96.653,-92.573,169.575,40.038,157.532
C09945=1037.946,96.902,-92.592,169.577,40.038,157.532
C09946=1037.953,97.151,-92.611,169.579,40.039,157.532
C09947=1037.959,97.401,-92.631,169.581,40.038,157.532
C09948=1037.965,97.650,-92.650,169.583,40.039,157.533
C09949=1037.971,97.899,-92.669,169.585,40.039,157.533
C09950=1037.977,98.148,-92.689,169.588,40.039,157.533
C09951=1037.984,98.397,-92.708,169.590,40.039,157.533
C09952=1037.990,98.646,-92.728,169.592,40.039,157.533
C09953=1037.997,98.896,-92.747,169.594,40.039,157.533
C09954=1038.002,99.145,-92.766,169.596,40.040,157.533
C09955=1038.009,99.394,-92.785,169.598,40.040,157.533
C09956=1038.015,99.643,-92.804,169.600,40.040,157.533
C09957=1038.022,99.892,-92.824,169.602,40.040,157.534
C09958=1038.028,100.142,-92.843,169.604,40.040,157.534
C09959=1038.035,100.390,-92.863,169.606,40.040,157.534
C09960=1038.040,100.640,-92.882,169.609,40.041,157.534
C09961=1038.046,100.889,-92.902,169.611,40.041,157.534
C09962=1038.052,101.138,-92.921,169.613,40.041,157.534
C09963=1038.059,101.388,-92.941,169.615,40.041,157.534
C09964=1038.065,101.637,-92.960,169.617,40.041,157.534
C09965=1038.071,101.886,-92.980,169.619,40.042,157.535
C09966=1038.077,102.135,-92.999,169.621,40.042,157.535
C09967=1038.083,102.384,-93.019,169.623,40.042,157.535
C09968=1038.089,102.634,-93.039,169.625,40.042,157.535
C09969=1038.096,102.882,-93.058,169.628,40.043,157.535
C09970=1038.102,103.131,-93.078,169.630,40.042,157.535
C09971=1038.107,103.381,-93.097,169.632,40.043,157.535
C09972=1038.113,103.629,-93.117,169.634,40.043,157.535
C09973=1038.120,103.879,-93.138,169.636,40.043,157.536
C09974=1038.126,104.128,-93.156,169.638,40.044,157.536
C09975=1038.132,104.377,-93.176,169.640,40.043,157.536
C09976=1038.138,104.626,-93.196,169.642,40.044,157.536
C09977=1038.145,104.876,-93.216,169.644,40.044,157.536
C09978=1038.151,105.125,-93.236,169.646,40.044,157.536
C09979=1038.157,105.374,-93.255,169.648,40.044,157.536
C09980=1038.163,105.623,-93.274,169.652,40.044,157.536
C09981=1038.170,105.872,-93.295,169.654,40.045,157.537
C09982=1038.175,106.122,-93.314,169.656,40.045,157.537
C09983=1038.181,106.370,-93.334,169.658,40.045,157.537
C09984=1038.189,106.620,-93.354,169.660,40.045,157.537
C09985=1038.194,106.869,-93.373,169.662,40.045,157.537
C09986=1038.200,107.118,-93.393,169.664,40.046,157.537
C09987=1038.206,107.367,-93.413,169.666,40.046,157.537
C09988=1038.213,107.616,-93.433,169.669,40.046,157.537
C09989=1038.219,107.866,-93.452,169.671,40.046,157.537
C09990=1038.225,108.114,-93.472,169.673,40.046,157.538
C09991=1038.232,108.364,-93.492,169.675,40.046,157.538
C09992=1038.239,108.650,-93.515,169.677,40.047,157.538
C09993=1038.246,108.935,-93.537,169.680,40.047,157.538
C09994=1038.253,109.221,-93.560,169.682,40.047,157.538
C09995=1038.260,109.507,-93.583,169.684,40.047,157.538
C09996=1038.267,109.757,-93.603,169.686,40.047,157.538
//INST
///DATE 2021/06/17 10:57
///ATTR SC,RW,RJ
////FRAME ROBOT
///GROUP1 RB1
NOP
MOVL C00000 V=800.0 PL=0
MOVL C00001 V=800.0 PL=0
MOVL C00002 V=800.0 PL=0
MOVL C00003 V=800.0 PL=0
MOVL C00004 V=800.0 PL=0
MOVL C00005 V=800.0 PL=0
MOVL C00006 V=800.0 PL=0
MOVL C00007 V=800.0 PL=0
MOVL C00008 V=800.0 PL=0
MOVL C00009 V=800.0 PL=0
MOVL C00010 V=800.0 PL=0
MOVL C00011 V=800.0 PL=0
MOVL C00012 V=800.0 PL=0
MOVL C00013 V=800.0 PL=0
MOVL C00014 V=800.0 PL=0
MOVL C00015 V=800.0 PL=0
MOVL C00016 V=800.0 PL=0
MOVL C00017 V=800.0 PL=0
MOVL C00018 V=800.0 PL=0
MOVL C00019 V=800.0 PL=0
MOVL C00020 V=800.0 PL=0
MOVL C00021 V=800.0 PL=0
MOVL C00022 V=800.0 PL=0
MOVL C00023 V=800.0 PL=0
MOVL C00024 V=800.0 PL=0
MOVL C00025 V=800.0 PL=0
MOVL C00026 V=800.0 PL=0
MOVL C00027 V=800.0 PL=0
MOVL C00028 V=800.0 PL=0
MOVL C00029 V=800.0 PL=0
MOVL C00030 V=800.0 PL=0
MOVL C00031 V=800.0 PL=0
MOVL C00032 V=800.0 PL=0
MOVL C00033 V=800.0 PL=0
MOVL C00034 V=800.0 PL=0
MOVL C00035 V=800.0 PL=0
MOVL C00036 V=800.0 PL=0
MOVL C00037 V=800.0 PL=0
MOVL C00038 V=800.0 PL=0
MOVL C00039 V=800.0 PL=0
MOVL C00040 V=800.0 PL=0
MOVL C00041 V=800.0 PL=0
MOVL C00042 V=800.0 PL=0
MOVL C00043 V=800.0 PL=0
MOVL C00044 V=800.0 PL=0
MOVL C00045 V=800.0 PL=0
MOVL C00046 V=800.0 PL=0
MOVL C00047 V=800.0 PL=0
MOVL C00048 V=800.0 PL=0
MOVL C00049 V=800.0 PL=0
MOVL C00050 V=800.0 PL=0
MOVL C00051 V=800.0 PL=0
MOVL C00052 V=800.0 PL=0
MOVL C00053 V=800.0 PL=0
MOVL C00054 V=800.0 PL=0
MOVL C00055 V=800.0 PL=0
MOVL C00056 V=800.0 PL=0
MOVL C00057 V=800.0 PL=0
MOVL C00058 V=800.0 PL=0
MOVL C00059 V=800.0 PL=0
MOVL C00060 V=800.0 PL=0
MOVL C00061 V=800.0 PL=0
MOVL C00062 V=800.0 PL=0
MOVL C00063 V=800.0 PL=0
MOVL C00064 V=800.0 PL=0
MOVL C00065 V=800.0 PL=0
MOVL C00066 V=800.0 PL=0
MOVL C00067 V=800.0 PL=0
MOVL C00068 V=800.0 PL=0
MOVL C00069 V=800.0 PL=0
MOVL C00070 V=800.0 PL=0
MOVL C00071 V=800.0 PL=0
MOVL C00072 V=800.0 PL=0
MOVL C00073 V=800.0 PL=0
MOVL C00074 V=800.0 PL=0
MOVL C00075 V=800.0 PL=0
MOVL C00076 V=800.0 PL=0
MOVL C00077 V=800.0 PL=0
MOVL C00078 V=800.0 PL=0
MOVL C00079 V=800.0 PL=0
MOVL C00080 V=800.0 PL=0
MOVL C00081 V=800.0 PL=0
MOVL C00082 V=800.0 PL=0
MOVL C00083 V=800.0 PL=0
MOVL C00084 V=800.0 PL=0
MOVL C00085 V=800.0 PL=0
MOVL C00086 V=800.0 PL=0
MOVL C00087 V=800.0 PL=0
MOVL C00088 V=800.0 PL=0
MOVL C00089 V=800.0 PL=0
MOVL C00090 V=800.0 PL=0
MOVL C00091 V=800.0 PL=0
MOVL C00092 V=800.0 PL=0
MOVL C00093 V=800.0 PL=0
MOVL C00094 V=800.0 PL=0
MOVL C00095 V=800.0 PL=0
MOVL C00096 V=800.0 PL=0
MOVL C00097 V=800.0 PL=0
MOVL C00098 V=800.0 PL=0
MOVL C00099 V=800.0 PL=0
MOVL C00100 V=800.0 PL=0
MOVL C00101 V=800.0 PL=0
MOVL C00102 V=800.0 PL=0
MOVL C00103 V=800.0 PL=0
MOVL C00104 V=800.0 PL=0
MOVL C00105 V=800.0 PL=0
MOVL C00106 V=800.0 PL=0
MOVL C00107 V=800.0 PL=0
MOVL C00108 V=800.0 PL=0
MOVL C00109 V=800.0 PL=0
MOVL C00110 V=800.0 PL=0
MOVL C00111 V=800.0 PL=0
MOVL C00112 V=800.0 PL=0
MOVL C00113 V=800.0 PL=0
MOVL C00114 V=800.0 PL=0
MOVL C00115 V=800.0 PL=0
MOVL C00116 V=800.0 PL=0
MOVL C00117 V=800.0 PL=0
MOVL C00118 V=800.0 PL=0
MOVL C00119 V=800.0 PL=0
MOVL C00120 V=800.0 PL=0
MOVL C00121 V=800.0 PL=0
MOVL C00122 V=800.0 PL=0
MOVL C00123 V=800.0 PL=0
MOVL C00124 V=800.0 PL=0
MOVL C00125 V=800.0 PL=0
MOVL C00126 V=800.0 PL=0
MOVL C00127 V=800.0 PL=0
MOVL C00128 V=800.0 PL=0
MOVL C00129 V=800.0 PL=0
MOVL C00130 V=800.0 PL=0
MOVL C00131 V=800.0 PL=0
MOVL C00132 V=800.0 PL=0
MOVL C00133 V=800.0 PL=0
MOVL C00134 V=800.0 PL=0
MOVL C00135 V=800.0 PL=0
MOVL C00136 V=800.0 PL=0
MOVL C00137 V=800.0 PL=0
MOVL C00138 V=800.0 PL=0
MOVL C00139 V=800.0 PL=0
MOVL C00140 V=800.0 PL=0
MOVL C00141 V=800.0 PL=0
MOVL C00142 V=800.0 PL=0
MOVL C00143 V=800.0 PL=0
MOVL C00144 V=800.0 PL=0
MOVL C00145 V=800.0 PL=0
MOVL C00146 V=800.0 PL=0
MOVL C00147 V=800.0 PL=0
MOVL C00148 V=800.0 PL=0
MOVL C00149 V=800.0 PL=0
MOVL C00150 V=800.0 PL=0
MOVL C00151 V=800.0 PL=0
MOVL C00152 V=800.0 PL=0
MOVL C00153 V=800.0 PL=0
MOVL C00154 V=800.0 PL=0
MOVL C00155 V=800.0 PL=0
MOVL C00156 V=800.0 PL=0
MOVL C00157 V=800.0 PL=0
MOVL C00158 V=800.0 PL=0
MOVL C00159 V=800.0 PL=0
MOVL C00160 V=800.0 PL=0
MOVL C00161 V=800.0 PL=0
MOVL C00162 V=800.0 PL=0
MOVL C00163 V=800.0 PL=0
MOVL C00164 V=800.0 PL=0
MOVL C00165 V=800.0 PL=0
MOVL C00166 V=800.0 PL=0
MOVL C00167 V=800.0 PL=0
MOVL C00168 V=800.0 PL=0
MOVL C00169 V=800.0 PL=0
MOVL C00170 V=800.0 PL=0
MOVL C00171 V=800.0 PL=0
MOVL C00172 V=800.0 PL=0
MOVL C00173 V=800.0 PL=0
MOVL C00174 V=800.0 PL=0
MOVL C00175 V=800.0 PL=0
MOVL C00176 V=800.0 PL=0
MOVL C00177 V=800.0 PL=0
MOVL C00178 V=800.0 PL=0
MOVL C00179 V=800.0 PL=0
MOVL C00180 V=800.0 PL=0
MOVL C00181 V=800.0 PL=0
MOVL C00182 V=800.0 PL=0
MOVL C00183 V=800.0 PL=0
MOVL C00184 V=800.0 PL=0
MOVL C00185 V=800.0 PL=0
MOVL C00186 V=800.0 PL=0
MOVL C00187 V=800.0 PL=0
MOVL C00188 V=800.0 PL=0
MOVL C00189 V=800.0 PL=0
MOVL C00190 V=800.0 PL=0
MOVL C00191 V=800.0 PL=0
MOVL C00192 V=800.0 PL=0
MOVL C00193 V=800.0 PL=0
MOVL C00194 V=800.0 PL=0
MOVL C00195 V=800.0 PL=0
MOVL C00196 V=800.0 PL=0
MOVL C00197 V=800.0 PL=0
MOVL C00198 V=800.0 PL=0
MOVL C00199 V=800.0 PL=0
MOVL C00200 V=800.0 PL=0
MOVL C00201 V=800.0 PL=0
MOVL C00202 V=800.0 PL=0
MOVL C00203 V=800.0 PL=0
MOVL C00204 V=800.0 PL=0
MOVL C00205 V=800.0 PL=0
MOVL C00206 V=800.0 PL=0
MOVL C00207 V=800.0 PL=0
MOVL C00208 V=800.0 PL=0
MOVL C00209 V=800.0 PL=0
MOVL C00210 V=800.0 PL=0
MOVL C00211 V=800.0 PL=0
MOVL C00212 V=800.0 PL=0
MOVL C00213 V=800.0 PL=0
MOVL C00214 V=800.0 PL=0
MOVL C00215 V=800.0 PL=0
MOVL C00216 V=800.0 PL=0
MOVL C00217 V=800.0 PL=0
MOVL C00218 V=800.0 PL=0
MOVL C00219 V=800.0 PL=0
MOVL C00220 V=800.0 PL=0
MOVL C00221 V=800.0 PL=0
MOVL C00222 V=800.0 PL=0
MOVL C00223 V=800.0 PL=0
MOVL C00224 V=800.0 PL=0
MOVL C00225 V=800.0 PL=0
MOVL C00226 V=800.0 PL=0
MOVL C00227 V=800.0 PL=0
MOVL C00228 V=800.0 PL=0
MOVL C00229 V=800.0 PL=0
MOVL C00230 V=800.0 PL=0
MOVL C00231 V=800.0 PL=0
MOVL C00232 V=800.0 PL=0
MOVL C00233 V=800.0 PL=0
MOVL C00234 V=800.0 PL=0
MOVL C00235 V=800.0 PL=0
MOVL C00236 V=800.0 PL=0
MOVL C00237 V=800.0 PL=0
MOVL C00238 V=800.0 PL=0
MOVL C00239 V=800.0 PL=0
MOVL C00240 V=800.0 PL=0
MOVL C00241 V=800.0 PL=0
MOVL C00242 V=800.0 PL=0
MOVL C00243 V=800.0 PL=0
MOVL C00244 V=800.0 PL=0
MOVL C00245 V=800.0 PL=0
MOVL C00246 V=800.0 PL=0
MOVL C00247 V=800.0 PL=0
MOVL C00248 V=800.0 PL=0
MOVL C00249 V=800.0 PL=0
MOVL C00250 V=800.0 PL=0
MOVL C00251 V=800.0 PL=0
MOVL C00252 V=800.0 PL=0
MOVL C00253 V=800.0 PL=0
MOVL C00254 V=800.0 PL=0
MOVL C00255 V=800.0 PL=0
MOVL C00256 V=800.0 PL=0
MOVL C00257 V=800.0 PL=0
MOVL C00258 V=800.0 PL=0
MOVL C00259 V=800.0 PL=0
MOVL C00260 V=800.0 PL=0
MOVL C00261 V=800.0 PL=0
MOVL C00262 V=800.0 PL=0
MOVL C00263 V=800.0 PL=0
MOVL C00264 V=800.0 PL=0
MOVL C00265 V=800.0 PL=0
MOVL C00266 V=800.0 PL=0
MOVL C00267 V=800.0 PL=0
MOVL C00268 V=800.0 PL=0
MOVL C00269 V=800.0 PL=0
MOVL C00270 V=800.0 PL=0
MOVL C00271 V=800.0 PL=0
MOVL C00272 V=800.0 PL=0
MOVL C00273 V=800.0 PL=0
MOVL C00274 V=800.0 PL=0
MOVL C00275 V=800.0 PL=0
MOVL C00276 V=800.0 PL=0
MOVL C00277 V=800.0 PL=0
MOVL C00278 V=800.0 PL=0
MOVL C00279 V=800.0 PL=0
MOVL C00280 V=800.0 PL=0
MOVL C00281 V=800.0 PL=0
MOVL C00282 V=800.0 PL=0
MOVL C00283 V=800.0 PL=0
MOVL C00284 V=800.0 PL=0
MOVL C00285 V=800.0 PL=0
MOVL C00286 V=800.0 PL=0
MOVL C00287 V=800.0 PL=0
MOVL C00288 V=800.0 PL=0
MOVL C00289 V=800.0 PL=0
MOVL C00290 V=800.0 PL=0
MOVL C00291 V=800.0 PL=0
MOVL C00292 V=800.0 PL=0
MOVL C00293 V=800.0 PL=0
MOVL C00294 V=800.0 PL=0
MOVL C00295 V=800.0 PL=0
MOVL C00296 V=800.0 PL=0
MOVL C00297 V=800.0 PL=0
MOVL C00298 V=800.0 PL=0
MOVL C00299 V=800.0 PL=0
MOVL C00300 V=800.0 PL=0
MOVL C00301 V=800.0 PL=0
MOVL C00302 V=800.0 PL=0
MOVL C00303 V=800.0 PL=0
MOVL C00304 V=800.0 PL=0
MOVL C00305 V=800.0 PL=0
MOVL C00306 V=800.0 PL=0
MOVL C00307 V=800.0 PL=0
MOVL C00308 V=800.0 PL=0
MOVL C00309 V=800.0 PL=0
MOVL C00310 V=800.0 PL=0
MOVL C00311 V=800.0 PL=0
MOVL C00312 V=800.0 PL=0
MOVL C00313 V=800.0 PL=0
MOVL C00314 V=800.0 PL=0
MOVL C00315 V=800.0 PL=0
MOVL C00316 V=800.0 PL=0
MOVL C00317 V=800.0 PL=0
MOVL C00318 V=800.0 PL=0
MOVL C00319 V=800.0 PL=0
MOVL C00320 V=800.0 PL=0
MOVL C00321 V=800.0 PL=0
MOVL C00322 V=800.0 PL=0
MOVL C00323 V=800.0 PL=0
MOVL C00324 V=800.0 PL=0
MOVL C00325 V=800.0 PL=0
MOVL C00326 V=800.0 PL=0
MOVL C00327 V=800.0 PL=0
MOVL C00328 V=800.0 PL=0
MOVL C00329 V=800.0 PL=0
MOVL C00330 V=800.0 PL=0
MOVL C00331 V=800.0 PL=0
MOVL C00332 V=800.0 PL=0
MOVL C00333 V=800.0 PL=0
MOVL C00334 V=800.0 PL=0
MOVL C00335 V=800.0 PL=0
MOVL C00336 V=800.0 PL=0
MOVL C00337 V=800.0 PL=0
MOVL C00338 V=800.0 PL=0
MOVL C00339 V=800.0 PL=0
MOVL C00340 V=800.0 PL=0
MOVL C00341 V=800.0 PL=0
MOVL C00342 V=800.0 PL=0
MOVL C00343 V=800.0 PL=0
MOVL C00344 V=800.0 PL=0
MOVL C00345 V=800.0 PL=0
MOVL C00346 V=800.0 PL=0
MOVL C00347 V=800.0 PL=0
MOVL C00348 V=800.0 PL=0
MOVL C00349 V=800.0 PL=0
MOVL C00350 V=800.0 PL=0
MOVL C00351 V=800.0 PL=0
MOVL C00352 V=800.0 PL=0
MOVL C00353 V=800.0 PL=0
MOVL C00354 V=800.0 PL=0
MOVL C00355 V=800.0 PL=0
MOVL C00356 V=800.0 PL=0
MOVL C00357 V=800.0 PL=0
MOVL C00358 V=800.0 PL=0
MOVL C00359 V=800.0 PL=0
MOVL C00360 V=800.0 PL=0
MOVL C00361 V=800.0 PL=0
MOVL C00362 V=800.0 PL=0
MOVL C00363 V=800.0 PL=0
MOVL C00364 V=800.0 PL=0
MOVL C00365 V=800.0 PL=0
MOVL C00366 V=800.0 PL=0
MOVL C00367 V=800.0 PL=0
MOVL C00368 V=800.0 PL=0
MOVL C00369 V=800.0 PL=0
MOVL C00370 V=800.0 PL=0
MOVL C00371 V=800.0 PL=0
MOVL C00372 V=800.0 PL=0
MOVL C00373 V=800.0 PL=0
MOVL C00374 V=800.0 PL=0
MOVL C00375 V=800.0 PL=0
MOVL C00376 V=800.0 PL=0
MOVL C00377 V=800.0 PL=0
MOVL C00378 V=800.0 PL=0
MOVL C00379 V=800.0 PL=0
MOVL C00380 V=800.0 PL=0
MOVL C00381 V=800.0 PL=0
MOVL C00382 V=800.0 PL=0
MOVL C00383 V=800.0 PL=0
MOVL C00384 V=800.0 PL=0
MOVL C00385 V=800.0 PL=0
MOVL C00386 V=800.0 PL=0
MOVL C00387 V=800.0 PL=0
MOVL C00388 V=800.0 PL=0
MOVL C00389 V=800.0 PL=0
MOVL C00390 V=800.0 PL=0
MOVL C00391 V=800.0 PL=0
MOVL C00392 V=800.0 PL=0
MOVL C00393 V=800.0 PL=0
MOVL C00394 V=800.0 PL=0
MOVL C00395 V=800.0 PL=0
MOVL C00396 V=800.0 PL=0
MOVL C00397 V=800.0 PL=0
MOVL C00398 V=800.0 PL=0
MOVL C00399 V=800.0 PL=0
MOVL C00400 V=800.0 PL=0
MOVL C00401 V=800.0 PL=0
MOVL C00402 V=800.0 PL=0
MOVL C00403 V=800.0 PL=0
MOVL C00404 V=800.0 PL=0
MOVL C00405 V=800.0 PL=0
MOVL C00406 V=800.0 PL=0
MOVL C00407 V=800.0 PL=0
MOVL C00408 V=800.0 PL=0
MOVL C00409 V=800.0 PL=0
MOVL C00410 V=800.0 PL=0
MOVL C00411 V=800.0 PL=0
MOVL C00412 V=800.0 PL=0
MOVL C00413 V=800.0 PL=0
MOVL C00414 V=800.0 PL=0
MOVL C00415 V=800.0 PL=0
MOVL C00416 V=800.0 PL=0
MOVL C00417 V=800.0 PL=0
MOVL C00418 V=800.0 PL=0
MOVL C00419 V=800.0 PL=0
MOVL C00420 V=800.0 PL=0
MOVL C00421 V=800.0 PL=0
MOVL C00422 V=800.0 PL=0
MOVL C00423 V=800.0 PL=0
MOVL C00424 V=800.0 PL=0
MOVL C00425 V=800.0 PL=0
MOVL C00426 V=800.0 PL=0
MOVL C00427 V=800.0 PL=0
MOVL C00428 V=800.0 PL=0
MOVL C00429 V=800.0 PL=0
MOVL C00430 V=800.0 PL=0
MOVL C00431 V=800.0 PL=0
MOVL C00432 V=800.0 PL=0
MOVL C00433 V=800.0 PL=0
MOVL C00434 V=800.0 PL=0
MOVL C00435 V=800.0 PL=0
MOVL C00436 V=800.0 PL=0
MOVL C00437 V=800.0 PL=0
MOVL C00438 V=800.0 PL=0
MOVL C00439 V=800.0 PL=0
MOVL C00440 V=800.0 PL=0
MOVL C00441 V=800.0 PL=0
MOVL C00442 V=800.0 PL=0
MOVL C00443 V=800.0 PL=0
MOVL C00444 V=800.0 PL=0
MOVL C00445 V=800.0 PL=0
MOVL C00446 V=800.0 PL=0
MOVL C00447 V=800.0 PL=0
MOVL C00448 V=800.0 PL=0
MOVL C00449 V=800.0 PL=0
MOVL C00450 V=800.0 PL=0
MOVL C00451 V=800.0 PL=0
MOVL C00452 V=800.0 PL=0
MOVL C00453 V=800.0 PL=0
MOVL C00454 V=800.0 PL=0
MOVL C00455 V=800.0 PL=0
MOVL C00456 V=800.0 PL=0
MOVL C00457 V=800.0 PL=0
MOVL C00458 V=800.0 PL=0
MOVL C00459 V=800.0 PL=0
MOVL C00460 V=800.0 PL=0
MOVL C00461 V=800.0 PL=0
MOVL C00462 V=800.0 PL=0
MOVL C00463 V=800.0 PL=0
MOVL C00464 V=800.0 PL=0
MOVL C00465 V=800.0 PL=0
MOVL C00466 V=800.0 PL=0
MOVL C00467 V=800.0 PL=0
MOVL C00468 V=800.0 PL=0
MOVL C00469 V=800.0 PL=0
MOVL C00470 V=800.0 PL=0
MOVL C00471 V=800.0 PL=0
MOVL C00472 V=800.0 PL=0
MOVL C00473 V=800.0 PL=0
MOVL C00474 V=800.0 PL=0
MOVL C00475 V=800.0 PL=0
MOVL C00476 V=800.0 PL=0
MOVL C00477 V=800.0 PL=0
MOVL C00478 V=800.0 PL=0
MOVL C00479 V=800.0 PL=0
MOVL C00480 V=800.0 PL=0
MOVL C00481 V=800.0 PL=0
MOVL C00482 V=800.0 PL=0
MOVL C00483 V=800.0 PL=0
MOVL C00484 V=800.0 PL=0
MOVL C00485 V=800.0 PL=0
MOVL C00486 V=800.0 PL=0
MOVL C00487 V=800.0 PL=0
MOVL C00488 V=800.0 PL=0
MOVL C00489 V=800.0 PL=0
MOVL C00490 V=800.0 PL=0
MOVL C00491 V=800.0 PL=0
MOVL C00492 V=800.0 PL=0
MOVL C00493 V=800.0 PL=0
MOVL C00494 V=800.0 PL=0
MOVL C00495 V=800.0 PL=0
MOVL C00496 V=800.0 PL=0
MOVL C00497 V=800.0 PL=0
MOVL C00498 V=800.0 PL=0
MOVL C00499 V=800.0 PL=0
MOVL C00500 V=800.0 PL=0
MOVL C00501 V=800.0 PL=0
MOVL C00502 V=800.0 PL=0
MOVL C00503 V=800.0 PL=0
MOVL C00504 V=800.0 PL=0
MOVL C00505 V=800.0 PL=0
MOVL C00506 V=800.0 PL=0
MOVL C00507 V=800.0 PL=0
MOVL C00508 V=800.0 PL=0
MOVL C00509 V=800.0 PL=0
MOVL C00510 V=800.0 PL=0
MOVL C00511 V=800.0 PL=0
MOVL C00512 V=800.0 PL=0
MOVL C00513 V=800.0 PL=0
MOVL C00514 V=800.0 PL=0
MOVL C00515 V=800.0 PL=0
MOVL C00516 V=800.0 PL=0
MOVL C00517 V=800.0 PL=0
MOVL C00518 V=800.0 PL=0
MOVL C00519 V=800.0 PL=0
MOVL C00520 V=800.0 PL=0
MOVL C00521 V=800.0 PL=0
MOVL C00522 V=800.0 PL=0
MOVL C00523 V=800.0 PL=0
MOVL C00524 V=800.0 PL=0
MOVL C00525 V=800.0 PL=0
MOVL C00526 V=800.0 PL=0
MOVL C00527 V=800.0 PL=0
MOVL C00528 V=800.0 PL=0
MOVL C00529 V=800.0 PL=0
MOVL C00530 V=800.0 PL=0
MOVL C00531 V=800.0 PL=0
MOVL C00532 V=800.0 PL=0
MOVL C00533 V=800.0 PL=0
MOVL C00534 V=800.0 PL=0
MOVL C00535 V=800.0 PL=0
MOVL C00536 V=800.0 PL=0
MOVL C00537 V=800.0 PL=0
MOVL C00538 V=800.0 PL=0
MOVL C00539 V=800.0 PL=0
MOVL C00540 V=800.0 PL=0
MOVL C00541 V=800.0 PL=0
MOVL C00542 V=800.0 PL=0
MOVL C00543 V=800.0 PL=0
MOVL C00544 V=800.0 PL=0
MOVL C00545 V=800.0 PL=0
MOVL C00546 V=800.0 PL=0
MOVL C00547 V=800.0 PL=0
MOVL C00548 V=800.0 PL=0
MOVL C00549 V=800.0 PL=0
MOVL C00550 V=800.0 PL=0
MOVL C00551 V=800.0 PL=0
MOVL C00552 V=800.0 PL=0
MOVL C00553 V=800.0 PL=0
MOVL C00554 V=800.0 PL=0
MOVL C00555 V=800.0 PL=0
MOVL C00556 V=800.0 PL=0
MOVL C00557 V=800.0 PL=0
MOVL C00558 V=800.0 PL=0
MOVL C00559 V=800.0 PL=0
MOVL C00560 V=800.0 PL=0
MOVL C00561 V=800.0 PL=0
MOVL C00562 V=800.0 PL=0
MOVL C00563 V=800.0 PL=0
MOVL C00564 V=800.0 PL=0
MOVL C00565 V=800.0 PL=0
MOVL C00566 V=800.0 PL=0
MOVL C00567 V=800.0 PL=0
MOVL C00568 V=800.0 PL=0
MOVL C00569 V=800.0 PL=0
MOVL C00570 V=800.0 PL=0
MOVL C00571 V=800.0 PL=0
MOVL C00572 V=800.0 PL=0
MOVL C00573 V=800.0 PL=0
MOVL C00574 V=800.0 PL=0
MOVL C00575 V=800.0 PL=0
MOVL C00576 V=800.0 PL=0
MOVL C00577 V=800.0 PL=0
MOVL C00578 V=800.0 PL=0
MOVL C00579 V=800.0 PL=0
MOVL C00580 V=800.0 PL=0
MOVL C00581 V=800.0 PL=0
MOVL C00582 V=800.0 PL=0
MOVL C00583 V=800.0 PL=0
MOVL C00584 V=800.0 PL=0
MOVL C00585 V=800.0 PL=0
MOVL C00586 V=800.0 PL=0
MOVL C00587 V=800.0 PL=0
MOVL C00588 V=800.0 PL=0
MOVL C00589 V=800.0 PL=0
MOVL C00590 V=800.0 PL=0
MOVL C00591 V=800.0 PL=0
MOVL C00592 V=800.0 PL=0
MOVL C00593 V=800.0 PL=0
MOVL C00594 V=800.0 PL=0
MOVL C00595 V=800.0 PL=0
MOVL C00596 V=800.0 PL=0
MOVL C00597 V=800.0 PL=0
MOVL C00598 V=800.0 PL=0
MOVL C00599 V=800.0 PL=0
MOVL C00600 V=800.0 PL=0
MOVL C00601 V=800.0 PL=0
MOVL C00602 V=800.0 PL=0
MOVL C00603 V=800.0 PL=0
MOVL C00604 V=800.0 PL=0
MOVL C00605 V=800.0 PL=0
MOVL C00606 V=800.0 PL=0
MOVL C00607 V=800.0 PL=0
MOVL C00608 V=800.0 PL=0
MOVL C00609 V=800.0 PL=0
MOVL C00610 V=800.0 PL=0
MOVL C00611 V=800.0 PL=0
MOVL C00612 V=800.0 PL=0
MOVL C00613 V=800.0 PL=0
MOVL C00614 V=800.0 PL=0
MOVL C00615 V=800.0 PL=0
MOVL C00616 V=800.0 PL=0
MOVL C00617 V=800.0 PL=0
MOVL C00618 V=800.0 PL=0
MOVL C00619 V=800.0 PL=0
MOVL C00620 V=800.0 PL=0
MOVL C00621 V=800.0 PL=0
MOVL C00622 V=800.0 PL=0
MOVL C00623 V=800.0 PL=0
MOVL C00624 V=800.0 PL=0
MOVL C00625 V=800.0 PL=0
MOVL C00626 V=800.0 PL=0
MOVL C00627 V=800.0 PL=0
MOVL C00628 V=800.0 PL=0
MOVL C00629 V=800.0 PL=0
MOVL C00630 V=800.0 PL=0
MOVL C00631 V=800.0 PL=0
MOVL C00632 V=800.0 PL=0
MOVL C00633 V=800.0 PL=0
MOVL C00634 V=800.0 PL=0
MOVL C00635 V=800.0 PL=0
MOVL C00636 V=800.0 PL=0
MOVL C00637 V=800.0 PL=0
MOVL C00638 V=800.0 PL=0
MOVL C00639 V=800.0 PL=0
MOVL C00640 V=800.0 PL=0
MOVL C00641 V=800.0 PL=0
MOVL C00642 V=800.0 PL=0
MOVL C00643 V=800.0 PL=0
MOVL C00644 V=800.0 PL=0
MOVL C00645 V=800.0 PL=0
MOVL C00646 V=800.0 PL=0
MOVL C00647 V=800.0 PL=0
MOVL C00648 V=800.0 PL=0
MOVL C00649 V=800.0 PL=0
MOVL C00650 V=800.0 PL=0
MOVL C00651 V=800.0 PL=0
MOVL C00652 V=800.0 PL=0
MOVL C00653 V=800.0 PL=0
MOVL C00654 V=800.0 PL=0
MOVL C00655 V=800.0 PL=0
MOVL C00656 V=800.0 PL=0
MOVL C00657 V=800.0 PL=0
MOVL C00658 V=800.0 PL=0
MOVL C00659 V=800.0 PL=0
MOVL C00660 V=800.0 PL=0
MOVL C00661 V=800.0 PL=0
MOVL C00662 V=800.0 PL=0
MOVL C00663 V=800.0 PL=0
MOVL C00664 V=800.0 PL=0
MOVL C00665 V=800.0 PL=0
MOVL C00666 V=800.0 PL=0
MOVL C00667 V=800.0 PL=0
MOVL C00668 V=800.0 PL=0
MOVL C00669 V=800.0 PL=0
MOVL C00670 V=800.0 PL=0
MOVL C00671 V=800.0 PL=0
MOVL C00672 V=800.0 PL=0
MOVL C00673 V=800.0 PL=0
MOVL C00674 V=800.0 PL=0
MOVL C00675 V=800.0 PL=0
MOVL C00676 V=800.0 PL=0
MOVL C00677 V=800.0 PL=0
MOVL C00678 V=800.0 PL=0
MOVL C00679 V=800.0 PL=0
MOVL C00680 V=800.0 PL=0
MOVL C00681 V=800.0 PL=0
MOVL C00682 V=800.0 PL=0
MOVL C00683 V=800.0 PL=0
MOVL C00684 V=800.0 PL=0
MOVL C00685 V=800.0 PL=0
MOVL C00686 V=800.0 PL=0
MOVL C00687 V=800.0 PL=0
MOVL C00688 V=800.0 PL=0
MOVL C00689 V=800.0 PL=0
MOVL C00690 V=800.0 PL=0
MOVL C00691 V=800.0 PL=0
MOVL C00692 V=800.0 PL=0
MOVL C00693 V=800.0 PL=0
MOVL C00694 V=800.0 PL=0
MOVL C00695 V=800.0 PL=0
MOVL C00696 V=800.0 PL=0
MOVL C00697 V=800.0 PL=0
MOVL C00698 V=800.0 PL=0
MOVL C00699 V=800.0 PL=0
MOVL C00700 V=800.0 PL=0
MOVL C00701 V=800.0 PL=0
MOVL C00702 V=800.0 PL=0
MOVL C00703 V=800.0 PL=0
MOVL C00704 V=800.0 PL=0
MOVL C00705 V=800.0 PL=0
MOVL C00706 V=800.0 PL=0
MOVL C00707 V=800.0 PL=0
MOVL C00708 V=800.0 PL=0
MOVL C00709 V=800.0 PL=0
MOVL C00710 V=800.0 PL=0
MOVL C00711 V=800.0 PL=0
MOVL C00712 V=800.0 PL=0
MOVL C00713 V=800.0 PL=0
MOVL C00714 V=800.0 PL=0
MOVL C00715 V=800.0 PL=0
MOVL C00716 V=800.0 PL=0
MOVL C00717 V=800.0 PL=0
MOVL C00718 V=800.0 PL=0
MOVL C00719 V=800.0 PL=0
MOVL C00720 V=800.0 PL=0
MOVL C00721 V=800.0 PL=0
MOVL C00722 V=800.0 PL=0
MOVL C00723 V=800.0 PL=0
MOVL C00724 V=800.0 PL=0
MOVL C00725 V=800.0 PL=0
MOVL C00726 V=800.0 PL=0
MOVL C00727 V=800.0 PL=0
MOVL C00728 V=800.0 PL=0
MOVL C00729 V=800.0 PL=0
MOVL C00730 V=800.0 PL=0
MOVL C00731 V=800.0 PL=0
MOVL C00732 V=800.0 PL=0
MOVL C00733 V=800.0 PL=0
MOVL C00734 V=800.0 PL=0
MOVL C00735 V=800.0 PL=0
MOVL C00736 V=800.0 PL=0
MOVL C00737 V=800.0 PL=0
MOVL C00738 V=800.0 PL=0
MOVL C00739 V=800.0 PL=0
MOVL C00740 V=800.0 PL=0
MOVL C00741 V=800.0 PL=0
MOVL C00742 V=800.0 PL=0
MOVL C00743 V=800.0 PL=0
MOVL C00744 V=800.0 PL=0
MOVL C00745 V=800.0 PL=0
MOVL C00746 V=800.0 PL=0
MOVL C00747 V=800.0 PL=0
MOVL C00748 V=800.0 PL=0
MOVL C00749 V=800.0 PL=0
MOVL C00750 V=800.0 PL=0
MOVL C00751 V=800.0 PL=0
MOVL C00752 V=800.0 PL=0
MOVL C00753 V=800.0 PL=0
MOVL C00754 V=800.0 PL=0
MOVL C00755 V=800.0 PL=0
MOVL C00756 V=800.0 PL=0
MOVL C00757 V=800.0 PL=0
MOVL C00758 V=800.0 PL=0
MOVL C00759 V=800.0 PL=0
MOVL C00760 V=800.0 PL=0
MOVL C00761 V=800.0 PL=0
MOVL C00762 V=800.0 PL=0
MOVL C00763 V=800.0 PL=0
MOVL C00764 V=800.0 PL=0
MOVL C00765 V=800.0 PL=0
MOVL C00766 V=800.0 PL=0
MOVL C00767 V=800.0 PL=0
MOVL C00768 V=800.0 PL=0
MOVL C00769 V=800.0 PL=0
MOVL C00770 V=800.0 PL=0
MOVL C00771 V=800.0 PL=0
MOVL C00772 V=800.0 PL=0
MOVL C00773 V=800.0 PL=0
MOVL C00774 V=800.0 PL=0
MOVL C00775 V=800.0 PL=0
MOVL C00776 V=800.0 PL=0
MOVL C00777 V=800.0 PL=0
MOVL C00778 V=800.0 PL=0
MOVL C00779 V=800.0 PL=0
MOVL C00780 V=800.0 PL=0
MOVL C00781 V=800.0 PL=0
MOVL C00782 V=800.0 PL=0
MOVL C00783 V=800.0 PL=0
MOVL C00784 V=800.0 PL=0
MOVL C00785 V=800.0 PL=0
MOVL C00786 V=800.0 PL=0
MOVL C00787 V=800.0 PL=0
MOVL C00788 V=800.0 PL=0
MOVL C00789 V=800.0 PL=0
MOVL C00790 V=800.0 PL=0
MOVL C00791 V=800.0 PL=0
MOVL C00792 V=800.0 PL=0
MOVL C00793 V=800.0 PL=0
MOVL C00794 V=800.0 PL=0
MOVL C00795 V=800.0 PL=0
MOVL C00796 V=800.0 PL=0
MOVL C00797 V=800.0 PL=0
MOVL C00798 V=800.0 PL=0
MOVL C00799 V=800.0 PL=0
MOVL C00800 V=800.0 PL=0
MOVL C00801 V=800.0 PL=0
MOVL C00802 V=800.0 PL=0
MOVL C00803 V=800.0 PL=0
MOVL C00804 V=800.0 PL=0
MOVL C00805 V=800.0 PL=0
MOVL C00806 V=800.0 PL=0
MOVL C00807 V=800.0 PL=0
MOVL C00808 V=800.0 PL=0
MOVL C00809 V=800.0 PL=0
MOVL C00810 V=800.0 PL=0
MOVL C00811 V=800.0 PL=0
MOVL C00812 V=800.0 PL=0
MOVL C00813 V=800.0 PL=0
MOVL C00814 V=800.0 PL=0
MOVL C00815 V=800.0 PL=0
MOVL C00816 V=800.0 PL=0
MOVL C00817 V=800.0 PL=0
MOVL C00818 V=800.0 PL=0
MOVL C00819 V=800.0 PL=0
MOVL C00820 V=800.0 PL=0
MOVL C00821 V=800.0 PL=0
MOVL C00822 V=800.0 PL=0
MOVL C00823 V=800.0 PL=0
MOVL C00824 V=800.0 PL=0
MOVL C00825 V=800.0 PL=0
MOVL C00826 V=800.0 PL=0
MOVL C00827 V=800.0 PL=0
MOVL C00828 V=800.0 PL=0
MOVL C00829 V=800.0 PL=0
MOVL C00830 V=800.0 PL=0
MOVL C00831 V=800.0 PL=0
MOVL C00832 V=800.0 PL=0
MOVL C00833 V=800.0 PL=0
MOVL C00834 V=800.0 PL=0
MOVL C00835 V=800.0 PL=0
MOVL C00836 V=800.0 PL=0
MOVL C00837 V=800.0 PL=0
MOVL C00838 V=800.0 PL=0
MOVL C00839 V=800.0 PL=0
MOVL C00840 V=800.0 PL=0
MOVL C00841 V=800.0 PL=0
MOVL C00842 V=800.0 PL=0
MOVL C00843 V=800.0 PL=0
MOVL C00844 V=800.0 PL=0
MOVL C00845 V=800.0 PL=0
MOVL C00846 V=800.0 PL=0
MOVL C00847 V=800.0 PL=0
MOVL C00848 V=800.0 PL=0
MOVL C00849 V=800.0 PL=0
MOVL C00850 V=800.0 PL=0
MOVL C00851 V=800.0 PL=0
MOVL C00852 V=800.0 PL=0
MOVL C00853 V=800.0 PL=0
MOVL C00854 V=800.0 PL=0
MOVL C00855 V=800.0 PL=0
MOVL C00856 V=800.0 PL=0
MOVL C00857 V=800.0 PL=0
MOVL C00858 V=800.0 PL=0
MOVL C00859 V=800.0 PL=0
MOVL C00860 V=800.0 PL=0
MOVL C00861 V=800.0 PL=0
MOVL C00862 V=800.0 PL=0
MOVL C00863 V=800.0 PL=0
MOVL C00864 V=800.0 PL=0
MOVL C00865 V=800.0 PL=0
MOVL C00866 V=800.0 PL=0
MOVL C00867 V=800.0 PL=0
MOVL C00868 V=800.0 PL=0
MOVL C00869 V=800.0 PL=0
MOVL C00870 V=800.0 PL=0
MOVL C00871 V=800.0 PL=0
MOVL C00872 V=800.0 PL=0
MOVL C00873 V=800.0 PL=0
MOVL C00874 V=800.0 PL=0
MOVL C00875 V=800.0 PL=0
MOVL C00876 V=800.0 PL=0
MOVL C00877 V=800.0 PL=0
MOVL C00878 V=800.0 PL=0
MOVL C00879 V=800.0 PL=0
MOVL C00880 V=800.0 PL=0
MOVL C00881 V=800.0 PL=0
MOVL C00882 V=800.0 PL=0
MOVL C00883 V=800.0 PL=0
MOVL C00884 V=800.0 PL=0
MOVL C00885 V=800.0 PL=0
MOVL C00886 V=800.0 PL=0
MOVL C00887 V=800.0 PL=0
MOVL C00888 V=800.0 PL=0
MOVL C00889 V=800.0 PL=0
MOVL C00890 V=800.0 PL=0
MOVL C00891 V=800.0 PL=0
MOVL C00892 V=800.0 PL=0
MOVL C00893 V=800.0 PL=0
MOVL C00894 V=800.0 PL=0
MOVL C00895 V=800.0 PL=0
MOVL C00896 V=800.0 PL=0
MOVL C00897 V=800.0 PL=0
MOVL C00898 V=800.0 PL=0
MOVL C00899 V=800.0 PL=0
MOVL C00900 V=800.0 PL=0
MOVL C00901 V=800.0 PL=0
MOVL C00902 V=800.0 PL=0
MOVL C00903 V=800.0 PL=0
MOVL C00904 V=800.0 PL=0
MOVL C00905 V=800.0 PL=0
MOVL C00906 V=800.0 PL=0
MOVL C00907 V=800.0 PL=0
MOVL C00908 V=800.0 PL=0
MOVL C00909 V=800.0 PL=0
MOVL C00910 V=800.0 PL=0
MOVL C00911 V=800.0 PL=0
MOVL C00912 V=800.0 PL=0
MOVL C00913 V=800.0 PL=0
MOVL C00914 V=800.0 PL=0
MOVL C00915 V=800.0 PL=0
MOVL C00916 V=800.0 PL=0
MOVL C00917 V=800.0 PL=0
MOVL C00918 V=800.0 PL=0
MOVL C00919 V=800.0 PL=0
MOVL C00920 V=800.0 PL=0
MOVL C00921 V=800.0 PL=0
MOVL C00922 V=800.0 PL=0
MOVL C00923 V=800.0 PL=0
MOVL C00924 V=800.0 PL=0
MOVL C00925 V=800.0 PL=0
MOVL C00926 V=800.0 PL=0
MOVL C00927 V=800.0 PL=0
MOVL C00928 V=800.0 PL=0
MOVL C00929 V=800.0 PL=0
MOVL C00930 V=800.0 PL=0
MOVL C00931 V=800.0 PL=0
MOVL C00932 V=800.0 PL=0
MOVL C00933 V=800.0 PL=0
MOVL C00934 V=800.0 PL=0
MOVL C00935 V=800.0 PL=0
MOVL C00936 V=800.0 PL=0
MOVL C00937 V=800.0 PL=0
MOVL C00938 V=800.0 PL=0
MOVL C00939 V=800.0 PL=0
MOVL C00940 V=800.0 PL=0
MOVL C00941 V=800.0 PL=0
MOVL C00942 V=800.0 PL=0
MOVL C00943 V=800.0 PL=0
MOVL C00944 V=800.0 PL=0
MOVL C00945 V=800.0 PL=0
MOVL C00946 V=800.0 PL=0
MOVL C00947 V=800.0 PL=0
MOVL C00948 V=800.0 PL=0
MOVL C00949 V=800.0 PL=0
MOVL C00950 V=800.0 PL=0
MOVL C00951 V=800.0 PL=0
MOVL C00952 V=800.0 PL=0
MOVL C00953 V=800.0 PL=0
MOVL C00954 V=800.0 PL=0
MOVL C00955 V=800.0 PL=0
MOVL C00956 V=800.0 PL=0
MOVL C00957 V=800.0 PL=0
MOVL C00958 V=800.0 PL=0
MOVL C00959 V=800.0 PL=0
MOVL C00960 V=800.0 PL=0
MOVL C00961 V=800.0 PL=0
MOVL C00962 V=800.0 PL=0
MOVL C00963 V=800.0 PL=0
MOVL C00964 V=800.0 PL=0
MOVL C00965 V=800.0 PL=0
MOVL C00966 V=800.0 PL=0
MOVL C00967 V=800.0 PL=0
MOVL C00968 V=800.0 PL=0
MOVL C00969 V=800.0 PL=0
MOVL C00970 V=800.0 PL=0
MOVL C00971 V=800.0 PL=0
MOVL C00972 V=800.0 PL=0
MOVL C00973 V=800.0 PL=0
MOVL C00974 V=800.0 PL=0
MOVL C00975 V=800.0 PL=0
MOVL C00976 V=800.0 PL=0
MOVL C00977 V=800.0 PL=0
MOVL C00978 V=800.0 PL=0
MOVL C00979 V=800.0 PL=0
MOVL C00980 V=800.0 PL=0
MOVL C00981 V=800.0 PL=0
MOVL C00982 V=800.0 PL=0
MOVL C00983 V=800.0 PL=0
MOVL C00984 V=800.0 PL=0
MOVL C00985 V=800.0 PL=0
MOVL C00986 V=800.0 PL=0
MOVL C00987 V=800.0 PL=0
MOVL C00988 V=800.0 PL=0
MOVL C00989 V=800.0 PL=0
MOVL C00990 V=800.0 PL=0
MOVL C00991 V=800.0 PL=0
MOVL C00992 V=800.0 PL=0
MOVL C00993 V=800.0 PL=0
MOVL C00994 V=800.0 PL=0
MOVL C00995 V=800.0 PL=0
MOVL C00996 V=800.0 PL=0
MOVL C00997 V=800.0 PL=0
MOVL C00998 V=800.0 PL=0
MOVL C00999 V=800.0 PL=0
MOVL C01000 V=800.0 PL=0
MOVL C01001 V=800.0 PL=0
MOVL C01002 V=800.0 PL=0
MOVL C01003 V=800.0 PL=0
MOVL C01004 V=800.0 PL=0
MOVL C01005 V=800.0 PL=0
MOVL C01006 V=800.0 PL=0
MOVL C01007 V=800.0 PL=0
MOVL C01008 V=800.0 PL=0
MOVL C01009 V=800.0 PL=0
MOVL C01010 V=800.0 PL=0
MOVL C01011 V=800.0 PL=0
MOVL C01012 V=800.0 PL=0
MOVL C01013 V=800.0 PL=0
MOVL C01014 V=800.0 PL=0
MOVL C01015 V=800.0 PL=0
MOVL C01016 V=800.0 PL=0
MOVL C01017 V=800.0 PL=0
MOVL C01018 V=800.0 PL=0
MOVL C01019 V=800.0 PL=0
MOVL C01020 V=800.0 PL=0
MOVL C01021 V=800.0 PL=0
MOVL C01022 V=800.0 PL=0
MOVL C01023 V=800.0 PL=0
MOVL C01024 V=800.0 PL=0
MOVL C01025 V=800.0 PL=0
MOVL C01026 V=800.0 PL=0
MOVL C01027 V=800.0 PL=0
MOVL C01028 V=800.0 PL=0
MOVL C01029 V=800.0 PL=0
MOVL C01030 V=800.0 PL=0
MOVL C01031 V=800.0 PL=0
MOVL C01032 V=800.0 PL=0
MOVL C01033 V=800.0 PL=0
MOVL C01034 V=800.0 PL=0
MOVL C01035 V=800.0 PL=0
MOVL C01036 V=800.0 PL=0
MOVL C01037 V=800.0 PL=0
MOVL C01038 V=800.0 PL=0
MOVL C01039 V=800.0 PL=0
MOVL C01040 V=800.0 PL=0
MOVL C01041 V=800.0 PL=0
MOVL C01042 V=800.0 PL=0
MOVL C01043 V=800.0 PL=0
MOVL C01044 V=800.0 PL=0
MOVL C01045 V=800.0 PL=0
MOVL C01046 V=800.0 PL=0
MOVL C01047 V=800.0 PL=0
MOVL C01048 V=800.0 PL=0
MOVL C01049 V=800.0 PL=0
MOVL C01050 V=800.0 PL=0
MOVL C01051 V=800.0 PL=0
MOVL C01052 V=800.0 PL=0
MOVL C01053 V=800.0 PL=0
MOVL C01054 V=800.0 PL=0
MOVL C01055 V=800.0 PL=0
MOVL C01056 V=800.0 PL=0
MOVL C01057 V=800.0 PL=0
MOVL C01058 V=800.0 PL=0
MOVL C01059 V=800.0 PL=0
MOVL C01060 V=800.0 PL=0
MOVL C01061 V=800.0 PL=0
MOVL C01062 V=800.0 PL=0
MOVL C01063 V=800.0 PL=0
MOVL C01064 V=800.0 PL=0
MOVL C01065 V=800.0 PL=0
MOVL C01066 V=800.0 PL=0
MOVL C01067 V=800.0 PL=0
MOVL C01068 V=800.0 PL=0
MOVL C01069 V=800.0 PL=0
MOVL C01070 V=800.0 PL=0
MOVL C01071 V=800.0 PL=0
MOVL C01072 V=800.0 PL=0
MOVL C01073 V=800.0 PL=0
MOVL C01074 V=800.0 PL=0
MOVL C01075 V=800.0 PL=0
MOVL C01076 V=800.0 PL=0
MOVL C01077 V=800.0 PL=0
MOVL C01078 V=800.0 PL=0
MOVL C01079 V=800.0 PL=0
MOVL C01080 V=800.0 PL=0
MOVL C01081 V=800.0 PL=0
MOVL C01082 V=800.0 PL=0
MOVL C01083 V=800.0 PL=0
MOVL C01084 V=800.0 PL=0
MOVL C01085 V=800.0 PL=0
MOVL C01086 V=800.0 PL=0
MOVL C01087 V=800.0 PL=0
MOVL C01088 V=800.0 PL=0
MOVL C01089 V=800.0 PL=0
MOVL C01090 V=800.0 PL=0
MOVL C01091 V=800.0 PL=0
MOVL C01092 V=800.0 PL=0
MOVL C01093 V=800.0 PL=0
MOVL C01094 V=800.0 PL=0
MOVL C01095 V=800.0 PL=0
MOVL C01096 V=800.0 PL=0
MOVL C01097 V=800.0 PL=0
MOVL C01098 V=800.0 PL=0
MOVL C01099 V=800.0 PL=0
MOVL C01100 V=800.0 PL=0
MOVL C01101 V=800.0 PL=0
MOVL C01102 V=800.0 PL=0
MOVL C01103 V=800.0 PL=0
MOVL C01104 V=800.0 PL=0
MOVL C01105 V=800.0 PL=0
MOVL C01106 V=800.0 PL=0
MOVL C01107 V=800.0 PL=0
MOVL C01108 V=800.0 PL=0
MOVL C01109 V=800.0 PL=0
MOVL C01110 V=800.0 PL=0
MOVL C01111 V=800.0 PL=0
MOVL C01112 V=800.0 PL=0
MOVL C01113 V=800.0 PL=0
MOVL C01114 V=800.0 PL=0
MOVL C01115 V=800.0 PL=0
MOVL C01116 V=800.0 PL=0
MOVL C01117 V=800.0 PL=0
MOVL C01118 V=800.0 PL=0
MOVL C01119 V=800.0 PL=0
MOVL C01120 V=800.0 PL=0
MOVL C01121 V=800.0 PL=0
MOVL C01122 V=800.0 PL=0
MOVL C01123 V=800.0 PL=0
MOVL C01124 V=800.0 PL=0
MOVL C01125 V=800.0 PL=0
MOVL C01126 V=800.0 PL=0
MOVL C01127 V=800.0 PL=0
MOVL C01128 V=800.0 PL=0
MOVL C01129 V=800.0 PL=0
MOVL C01130 V=800.0 PL=0
MOVL C01131 V=800.0 PL=0
MOVL C01132 V=800.0 PL=0
MOVL C01133 V=800.0 PL=0
MOVL C01134 V=800.0 PL=0
MOVL C01135 V=800.0 PL=0
MOVL C01136 V=800.0 PL=0
MOVL C01137 V=800.0 PL=0
MOVL C01138 V=800.0 PL=0
MOVL C01139 V=800.0 PL=0
MOVL C01140 V=800.0 PL=0
MOVL C01141 V=800.0 PL=0
MOVL C01142 V=800.0 PL=0
MOVL C01143 V=800.0 PL=0
MOVL C01144 V=800.0 PL=0
MOVL C01145 V=800.0 PL=0
MOVL C01146 V=800.0 PL=0
MOVL C01147 V=800.0 PL=0
MOVL C01148 V=800.0 PL=0
MOVL C01149 V=800.0 PL=0
MOVL C01150 V=800.0 PL=0
MOVL C01151 V=800.0 PL=0
MOVL C01152 V=800.0 PL=0
MOVL C01153 V=800.0 PL=0
MOVL C01154 V=800.0 PL=0
MOVL C01155 V=800.0 PL=0
MOVL C01156 V=800.0 PL=0
MOVL C01157 V=800.0 PL=0
MOVL C01158 V=800.0 PL=0
MOVL C01159 V=800.0 PL=0
MOVL C01160 V=800.0 PL=0
MOVL C01161 V=800.0 PL=0
MOVL C01162 V=800.0 PL=0
MOVL C01163 V=800.0 PL=0
MOVL C01164 V=800.0 PL=0
MOVL C01165 V=800.0 PL=0
MOVL C01166 V=800.0 PL=0
MOVL C01167 V=800.0 PL=0
MOVL C01168 V=800.0 PL=0
MOVL C01169 V=800.0 PL=0
MOVL C01170 V=800.0 PL=0
MOVL C01171 V=800.0 PL=0
MOVL C01172 V=800.0 PL=0
MOVL C01173 V=800.0 PL=0
MOVL C01174 V=800.0 PL=0
MOVL C01175 V=800.0 PL=0
MOVL C01176 V=800.0 PL=0
MOVL C01177 V=800.0 PL=0
MOVL C01178 V=800.0 PL=0
MOVL C01179 V=800.0 PL=0
MOVL C01180 V=800.0 PL=0
MOVL C01181 V=800.0 PL=0
MOVL C01182 V=800.0 PL=0
MOVL C01183 V=800.0 PL=0
MOVL C01184 V=800.0 PL=0
MOVL C01185 V=800.0 PL=0
MOVL C01186 V=800.0 PL=0
MOVL C01187 V=800.0 PL=0
MOVL C01188 V=800.0 PL=0
MOVL C01189 V=800.0 PL=0
MOVL C01190 V=800.0 PL=0
MOVL C01191 V=800.0 PL=0
MOVL C01192 V=800.0 PL=0
MOVL C01193 V=800.0 PL=0
MOVL C01194 V=800.0 PL=0
MOVL C01195 V=800.0 PL=0
MOVL C01196 V=800.0 PL=0
MOVL C01197 V=800.0 PL=0
MOVL C01198 V=800.0 PL=0
MOVL C01199 V=800.0 PL=0
MOVL C01200 V=800.0 PL=0
MOVL C01201 V=800.0 PL=0
MOVL C01202 V=800.0 PL=0
MOVL C01203 V=800.0 PL=0
MOVL C01204 V=800.0 PL=0
MOVL C01205 V=800.0 PL=0
MOVL C01206 V=800.0 PL=0
MOVL C01207 V=800.0 PL=0
MOVL C01208 V=800.0 PL=0
MOVL C01209 V=800.0 PL=0
MOVL C01210 V=800.0 PL=0
MOVL C01211 V=800.0 PL=0
MOVL C01212 V=800.0 PL=0
MOVL C01213 V=800.0 PL=0
MOVL C01214 V=800.0 PL=0
MOVL C01215 V=800.0 PL=0
MOVL C01216 V=800.0 PL=0
MOVL C01217 V=800.0 PL=0
MOVL C01218 V=800.0 PL=0
MOVL C01219 V=800.0 PL=0
MOVL C01220 V=800.0 PL=0
MOVL C01221 V=800.0 PL=0
MOVL C01222 V=800.0 PL=0
MOVL C01223 V=800.0 PL=0
MOVL C01224 V=800.0 PL=0
MOVL C01225 V=800.0 PL=0
MOVL C01226 V=800.0 PL=0
MOVL C01227 V=800.0 PL=0
MOVL C01228 V=800.0 PL=0
MOVL C01229 V=800.0 PL=0
MOVL C01230 V=800.0 PL=0
MOVL C01231 V=800.0 PL=0
MOVL C01232 V=800.0 PL=0
MOVL C01233 V=800.0 PL=0
MOVL C01234 V=800.0 PL=0
MOVL C01235 V=800.0 PL=0
MOVL C01236 V=800.0 PL=0
MOVL C01237 V=800.0 PL=0
MOVL C01238 V=800.0 PL=0
MOVL C01239 V=800.0 PL=0
MOVL C01240 V=800.0 PL=0
MOVL C01241 V=800.0 PL=0
MOVL C01242 V=800.0 PL=0
MOVL C01243 V=800.0 PL=0
MOVL C01244 V=800.0 PL=0
MOVL C01245 V=800.0 PL=0
MOVL C01246 V=800.0 PL=0
MOVL C01247 V=800.0 PL=0
MOVL C01248 V=800.0 PL=0
MOVL C01249 V=800.0 PL=0
MOVL C01250 V=800.0 PL=0
MOVL C01251 V=800.0 PL=0
MOVL C01252 V=800.0 PL=0
MOVL C01253 V=800.0 PL=0
MOVL C01254 V=800.0 PL=0
MOVL C01255 V=800.0 PL=0
MOVL C01256 V=800.0 PL=0
MOVL C01257 V=800.0 PL=0
MOVL C01258 V=800.0 PL=0
MOVL C01259 V=800.0 PL=0
MOVL C01260 V=800.0 PL=0
MOVL C01261 V=800.0 PL=0
MOVL C01262 V=800.0 PL=0
MOVL C01263 V=800.0 PL=0
MOVL C01264 V=800.0 PL=0
MOVL C01265 V=800.0 PL=0
MOVL C01266 V=800.0 PL=0
MOVL C01267 V=800.0 PL=0
MOVL C01268 V=800.0 PL=0
MOVL C01269 V=800.0 PL=0
MOVL C01270 V=800.0 PL=0
MOVL C01271 V=800.0 PL=0
MOVL C01272 V=800.0 PL=0
MOVL C01273 V=800.0 PL=0
MOVL C01274 V=800.0 PL=0
MOVL C01275 V=800.0 PL=0
MOVL C01276 V=800.0 PL=0
MOVL C01277 V=800.0 PL=0
MOVL C01278 V=800.0 PL=0
MOVL C01279 V=800.0 PL=0
MOVL C01280 V=800.0 PL=0
MOVL C01281 V=800.0 PL=0
MOVL C01282 V=800.0 PL=0
MOVL C01283 V=800.0 PL=0
MOVL C01284 V=800.0 PL=0
MOVL C01285 V=800.0 PL=0
MOVL C01286 V=800.0 PL=0
MOVL C01287 V=800.0 PL=0
MOVL C01288 V=800.0 PL=0
MOVL C01289 V=800.0 PL=0
MOVL C01290 V=800.0 PL=0
MOVL C01291 V=800.0 PL=0
MOVL C01292 V=800.0 PL=0
MOVL C01293 V=800.0 PL=0
MOVL C01294 V=800.0 PL=0
MOVL C01295 V=800.0 PL=0
MOVL C01296 V=800.0 PL=0
MOVL C01297 V=800.0 PL=0
MOVL C01298 V=800.0 PL=0
MOVL C01299 V=800.0 PL=0
MOVL C01300 V=800.0 PL=0
MOVL C01301 V=800.0 PL=0
MOVL C01302 V=800.0 PL=0
MOVL C01303 V=800.0 PL=0
MOVL C01304 V=800.0 PL=0
MOVL C01305 V=800.0 PL=0
MOVL C01306 V=800.0 PL=0
MOVL C01307 V=800.0 PL=0
MOVL C01308 V=800.0 PL=0
MOVL C01309 V=800.0 PL=0
MOVL C01310 V=800.0 PL=0
MOVL C01311 V=800.0 PL=0
MOVL C01312 V=800.0 PL=0
MOVL C01313 V=800.0 PL=0
MOVL C01314 V=800.0 PL=0
MOVL C01315 V=800.0 PL=0
MOVL C01316 V=800.0 PL=0
MOVL C01317 V=800.0 PL=0
MOVL C01318 V=800.0 PL=0
MOVL C01319 V=800.0 PL=0
MOVL C01320 V=800.0 PL=0
MOVL C01321 V=800.0 PL=0
MOVL C01322 V=800.0 PL=0
MOVL C01323 V=800.0 PL=0
MOVL C01324 V=800.0 PL=0
MOVL C01325 V=800.0 PL=0
MOVL C01326 V=800.0 PL=0
MOVL C01327 V=800.0 PL=0
MOVL C01328 V=800.0 PL=0
MOVL C01329 V=800.0 PL=0
MOVL C01330 V=800.0 PL=0
MOVL C01331 V=800.0 PL=0
MOVL C01332 V=800.0 PL=0
MOVL C01333 V=800.0 PL=0
MOVL C01334 V=800.0 PL=0
MOVL C01335 V=800.0 PL=0
MOVL C01336 V=800.0 PL=0
MOVL C01337 V=800.0 PL=0
MOVL C01338 V=800.0 PL=0
MOVL C01339 V=800.0 PL=0
MOVL C01340 V=800.0 PL=0
MOVL C01341 V=800.0 PL=0
MOVL C01342 V=800.0 PL=0
MOVL C01343 V=800.0 PL=0
MOVL C01344 V=800.0 PL=0
MOVL C01345 V=800.0 PL=0
MOVL C01346 V=800.0 PL=0
MOVL C01347 V=800.0 PL=0
MOVL C01348 V=800.0 PL=0
MOVL C01349 V=800.0 PL=0
MOVL C01350 V=800.0 PL=0
MOVL C01351 V=800.0 PL=0
MOVL C01352 V=800.0 PL=0
MOVL C01353 V=800.0 PL=0
MOVL C01354 V=800.0 PL=0
MOVL C01355 V=800.0 PL=0
MOVL C01356 V=800.0 PL=0
MOVL C01357 V=800.0 PL=0
MOVL C01358 V=800.0 PL=0
MOVL C01359 V=800.0 PL=0
MOVL C01360 V=800.0 PL=0
MOVL C01361 V=800.0 PL=0
MOVL C01362 V=800.0 PL=0
MOVL C01363 V=800.0 PL=0
MOVL C01364 V=800.0 PL=0
MOVL C01365 V=800.0 PL=0
MOVL C01366 V=800.0 PL=0
MOVL C01367 V=800.0 PL=0
MOVL C01368 V=800.0 PL=0
MOVL C01369 V=800.0 PL=0
MOVL C01370 V=800.0 PL=0
MOVL C01371 V=800.0 PL=0
MOVL C01372 V=800.0 PL=0
MOVL C01373 V=800.0 PL=0
MOVL C01374 V=800.0 PL=0
MOVL C01375 V=800.0 PL=0
MOVL C01376 V=800.0 PL=0
MOVL C01377 V=800.0 PL=0
MOVL C01378 V=800.0 PL=0
MOVL C01379 V=800.0 PL=0
MOVL C01380 V=800.0 PL=0
MOVL C01381 V=800.0 PL=0
MOVL C01382 V=800.0 PL=0
MOVL C01383 V=800.0 PL=0
MOVL C01384 V=800.0 PL=0
MOVL C01385 V=800.0 PL=0
MOVL C01386 V=800.0 PL=0
MOVL C01387 V=800.0 PL=0
MOVL C01388 V=800.0 PL=0
MOVL C01389 V=800.0 PL=0
MOVL C01390 V=800.0 PL=0
MOVL C01391 V=800.0 PL=0
MOVL C01392 V=800.0 PL=0
MOVL C01393 V=800.0 PL=0
MOVL C01394 V=800.0 PL=0
MOVL C01395 V=800.0 PL=0
MOVL C01396 V=800.0 PL=0
MOVL C01397 V=800.0 PL=0
MOVL C01398 V=800.0 PL=0
MOVL C01399 V=800.0 PL=0
MOVL C01400 V=800.0 PL=0
MOVL C01401 V=800.0 PL=0
MOVL C01402 V=800.0 PL=0
MOVL C01403 V=800.0 PL=0
MOVL C01404 V=800.0 PL=0
MOVL C01405 V=800.0 PL=0
MOVL C01406 V=800.0 PL=0
MOVL C01407 V=800.0 PL=0
MOVL C01408 V=800.0 PL=0
MOVL C01409 V=800.0 PL=0
MOVL C01410 V=800.0 PL=0
MOVL C01411 V=800.0 PL=0
MOVL C01412 V=800.0 PL=0
MOVL C01413 V=800.0 PL=0
MOVL C01414 V=800.0 PL=0
MOVL C01415 V=800.0 PL=0
MOVL C01416 V=800.0 PL=0
MOVL C01417 V=800.0 PL=0
MOVL C01418 V=800.0 PL=0
MOVL C01419 V=800.0 PL=0
MOVL C01420 V=800.0 PL=0
MOVL C01421 V=800.0 PL=0
MOVL C01422 V=800.0 PL=0
MOVL C01423 V=800.0 PL=0
MOVL C01424 V=800.0 PL=0
MOVL C01425 V=800.0 PL=0
MOVL C01426 V=800.0 PL=0
MOVL C01427 V=800.0 PL=0
MOVL C01428 V=800.0 PL=0
MOVL C01429 V=800.0 PL=0
MOVL C01430 V=800.0 PL=0
MOVL C01431 V=800.0 PL=0
MOVL C01432 V=800.0 PL=0
MOVL C01433 V=800.0 PL=0
MOVL C01434 V=800.0 PL=0
MOVL C01435 V=800.0 PL=0
MOVL C01436 V=800.0 PL=0
MOVL C01437 V=800.0 PL=0
MOVL C01438 V=800.0 PL=0
MOVL C01439 V=800.0 PL=0
MOVL C01440 V=800.0 PL=0
MOVL C01441 V=800.0 PL=0
MOVL C01442 V=800.0 PL=0
MOVL C01443 V=800.0 PL=0
MOVL C01444 V=800.0 PL=0
MOVL C01445 V=800.0 PL=0
MOVL C01446 V=800.0 PL=0
MOVL C01447 V=800.0 PL=0
MOVL C01448 V=800.0 PL=0
MOVL C01449 V=800.0 PL=0
MOVL C01450 V=800.0 PL=0
MOVL C01451 V=800.0 PL=0
MOVL C01452 V=800.0 PL=0
MOVL C01453 V=800.0 PL=0
MOVL C01454 V=800.0 PL=0
MOVL C01455 V=800.0 PL=0
MOVL C01456 V=800.0 PL=0
MOVL C01457 V=800.0 PL=0
MOVL C01458 V=800.0 PL=0
MOVL C01459 V=800.0 PL=0
MOVL C01460 V=800.0 PL=0
MOVL C01461 V=800.0 PL=0
MOVL C01462 V=800.0 PL=0
MOVL C01463 V=800.0 PL=0
MOVL C01464 V=800.0 PL=0
MOVL C01465 V=800.0 PL=0
MOVL C01466 V=800.0 PL=0
MOVL C01467 V=800.0 PL=0
MOVL C01468 V=800.0 PL=0
MOVL C01469 V=800.0 PL=0
MOVL C01470 V=800.0 PL=0
MOVL C01471 V=800.0 PL=0
MOVL C01472 V=800.0 PL=0
MOVL C01473 V=800.0 PL=0
MOVL C01474 V=800.0 PL=0
MOVL C01475 V=800.0 PL=0
MOVL C01476 V=800.0 PL=0
MOVL C01477 V=800.0 PL=0
MOVL C01478 V=800.0 PL=0
MOVL C01479 V=800.0 PL=0
MOVL C01480 V=800.0 PL=0
MOVL C01481 V=800.0 PL=0
MOVL C01482 V=800.0 PL=0
MOVL C01483 V=800.0 PL=0
MOVL C01484 V=800.0 PL=0
MOVL C01485 V=800.0 PL=0
MOVL C01486 V=800.0 PL=0
MOVL C01487 V=800.0 PL=0
MOVL C01488 V=800.0 PL=0
MOVL C01489 V=800.0 PL=0
MOVL C01490 V=800.0 PL=0
MOVL C01491 V=800.0 PL=0
MOVL C01492 V=800.0 PL=0
MOVL C01493 V=800.0 PL=0
MOVL C01494 V=800.0 PL=0
MOVL C01495 V=800.0 PL=0
MOVL C01496 V=800.0 PL=0
MOVL C01497 V=800.0 PL=0
MOVL C01498 V=800.0 PL=0
MOVL C01499 V=800.0 PL=0
MOVL C01500 V=800.0 PL=0
MOVL C01501 V=800.0 PL=0
MOVL C01502 V=800.0 PL=0
MOVL C01503 V=800.0 PL=0
MOVL C01504 V=800.0 PL=0
MOVL C01505 V=800.0 PL=0
MOVL C01506 V=800.0 PL=0
MOVL C01507 V=800.0 PL=0
MOVL C01508 V=800.0 PL=0
MOVL C01509 V=800.0 PL=0
MOVL C01510 V=800.0 PL=0
MOVL C01511 V=800.0 PL=0
MOVL C01512 V=800.0 PL=0
MOVL C01513 V=800.0 PL=0
MOVL C01514 V=800.0 PL=0
MOVL C01515 V=800.0 PL=0
MOVL C01516 V=800.0 PL=0
MOVL C01517 V=800.0 PL=0
MOVL C01518 V=800.0 PL=0
MOVL C01519 V=800.0 PL=0
MOVL C01520 V=800.0 PL=0
MOVL C01521 V=800.0 PL=0
MOVL C01522 V=800.0 PL=0
MOVL C01523 V=800.0 PL=0
MOVL C01524 V=800.0 PL=0
MOVL C01525 V=800.0 PL=0
MOVL C01526 V=800.0 PL=0
MOVL C01527 V=800.0 PL=0
MOVL C01528 V=800.0 PL=0
MOVL C01529 V=800.0 PL=0
MOVL C01530 V=800.0 PL=0
MOVL C01531 V=800.0 PL=0
MOVL C01532 V=800.0 PL=0
MOVL C01533 V=800.0 PL=0
MOVL C01534 V=800.0 PL=0
MOVL C01535 V=800.0 PL=0
MOVL C01536 V=800.0 PL=0
MOVL C01537 V=800.0 PL=0
MOVL C01538 V=800.0 PL=0
MOVL C01539 V=800.0 PL=0
MOVL C01540 V=800.0 PL=0
MOVL C01541 V=800.0 PL=0
MOVL C01542 V=800.0 PL=0
MOVL C01543 V=800.0 PL=0
MOVL C01544 V=800.0 PL=0
MOVL C01545 V=800.0 PL=0
MOVL C01546 V=800.0 PL=0
MOVL C01547 V=800.0 PL=0
MOVL C01548 V=800.0 PL=0
MOVL C01549 V=800.0 PL=0
MOVL C01550 V=800.0 PL=0
MOVL C01551 V=800.0 PL=0
MOVL C01552 V=800.0 PL=0
MOVL C01553 V=800.0 PL=0
MOVL C01554 V=800.0 PL=0
MOVL C01555 V=800.0 PL=0
MOVL C01556 V=800.0 PL=0
MOVL C01557 V=800.0 PL=0
MOVL C01558 V=800.0 PL=0
MOVL C01559 V=800.0 PL=0
MOVL C01560 V=800.0 PL=0
MOVL C01561 V=800.0 PL=0
MOVL C01562 V=800.0 PL=0
MOVL C01563 V=800.0 PL=0
MOVL C01564 V=800.0 PL=0
MOVL C01565 V=800.0 PL=0
MOVL C01566 V=800.0 PL=0
MOVL C01567 V=800.0 PL=0
MOVL C01568 V=800.0 PL=0
MOVL C01569 V=800.0 PL=0
MOVL C01570 V=800.0 PL=0
MOVL C01571 V=800.0 PL=0
MOVL C01572 V=800.0 PL=0
MOVL C01573 V=800.0 PL=0
MOVL C01574 V=800.0 PL=0
MOVL C01575 V=800.0 PL=0
MOVL C01576 V=800.0 PL=0
MOVL C01577 V=800.0 PL=0
MOVL C01578 V=800.0 PL=0
MOVL C01579 V=800.0 PL=0
MOVL C01580 V=800.0 PL=0
MOVL C01581 V=800.0 PL=0
MOVL C01582 V=800.0 PL=0
MOVL C01583 V=800.0 PL=0
MOVL C01584 V=800.0 PL=0
MOVL C01585 V=800.0 PL=0
MOVL C01586 V=800.0 PL=0
MOVL C01587 V=800.0 PL=0
MOVL C01588 V=800.0 PL=0
MOVL C01589 V=800.0 PL=0
MOVL C01590 V=800.0 PL=0
MOVL C01591 V=800.0 PL=0
MOVL C01592 V=800.0 PL=0
MOVL C01593 V=800.0 PL=0
MOVL C01594 V=800.0 PL=0
MOVL C01595 V=800.0 PL=0
MOVL C01596 V=800.0 PL=0
MOVL C01597 V=800.0 PL=0
MOVL C01598 V=800.0 PL=0
MOVL C01599 V=800.0 PL=0
MOVL C01600 V=800.0 PL=0
MOVL C01601 V=800.0 PL=0
MOVL C01602 V=800.0 PL=0
MOVL C01603 V=800.0 PL=0
MOVL C01604 V=800.0 PL=0
MOVL C01605 V=800.0 PL=0
MOVL C01606 V=800.0 PL=0
MOVL C01607 V=800.0 PL=0
MOVL C01608 V=800.0 PL=0
MOVL C01609 V=800.0 PL=0
MOVL C01610 V=800.0 PL=0
MOVL C01611 V=800.0 PL=0
MOVL C01612 V=800.0 PL=0
MOVL C01613 V=800.0 PL=0
MOVL C01614 V=800.0 PL=0
MOVL C01615 V=800.0 PL=0
MOVL C01616 V=800.0 PL=0
MOVL C01617 V=800.0 PL=0
MOVL C01618 V=800.0 PL=0
MOVL C01619 V=800.0 PL=0
MOVL C01620 V=800.0 PL=0
MOVL C01621 V=800.0 PL=0
MOVL C01622 V=800.0 PL=0
MOVL C01623 V=800.0 PL=0
MOVL C01624 V=800.0 PL=0
MOVL C01625 V=800.0 PL=0
MOVL C01626 V=800.0 PL=0
MOVL C01627 V=800.0 PL=0
MOVL C01628 V=800.0 PL=0
MOVL C01629 V=800.0 PL=0
MOVL C01630 V=800.0 PL=0
MOVL C01631 V=800.0 PL=0
MOVL C01632 V=800.0 PL=0
MOVL C01633 V=800.0 PL=0
MOVL C01634 V=800.0 PL=0
MOVL C01635 V=800.0 PL=0
MOVL C01636 V=800.0 PL=0
MOVL C01637 V=800.0 PL=0
MOVL C01638 V=800.0 PL=0
MOVL C01639 V=800.0 PL=0
MOVL C01640 V=800.0 PL=0
MOVL C01641 V=800.0 PL=0
MOVL C01642 V=800.0 PL=0
MOVL C01643 V=800.0 PL=0
MOVL C01644 V=800.0 PL=0
MOVL C01645 V=800.0 PL=0
MOVL C01646 V=800.0 PL=0
MOVL C01647 V=800.0 PL=0
MOVL C01648 V=800.0 PL=0
MOVL C01649 V=800.0 PL=0
MOVL C01650 V=800.0 PL=0
MOVL C01651 V=800.0 PL=0
MOVL C01652 V=800.0 PL=0
MOVL C01653 V=800.0 PL=0
MOVL C01654 V=800.0 PL=0
MOVL C01655 V=800.0 PL=0
MOVL C01656 V=800.0 PL=0
MOVL C01657 V=800.0 PL=0
MOVL C01658 V=800.0 PL=0
MOVL C01659 V=800.0 PL=0
MOVL C01660 V=800.0 PL=0
MOVL C01661 V=800.0 PL=0
MOVL C01662 V=800.0 PL=0
MOVL C01663 V=800.0 PL=0
MOVL C01664 V=800.0 PL=0
MOVL C01665 V=800.0 PL=0
MOVL C01666 V=800.0 PL=0
MOVL C01667 V=800.0 PL=0
MOVL C01668 V=800.0 PL=0
MOVL C01669 V=800.0 PL=0
MOVL C01670 V=800.0 PL=0
MOVL C01671 V=800.0 PL=0
MOVL C01672 V=800.0 PL=0
MOVL C01673 V=800.0 PL=0
MOVL C01674 V=800.0 PL=0
MOVL C01675 V=800.0 PL=0
MOVL C01676 V=800.0 PL=0
MOVL C01677 V=800.0 PL=0
MOVL C01678 V=800.0 PL=0
MOVL C01679 V=800.0 PL=0
MOVL C01680 V=800.0 PL=0
MOVL C01681 V=800.0 PL=0
MOVL C01682 V=800.0 PL=0
MOVL C01683 V=800.0 PL=0
MOVL C01684 V=800.0 PL=0
MOVL C01685 V=800.0 PL=0
MOVL C01686 V=800.0 PL=0
MOVL C01687 V=800.0 PL=0
MOVL C01688 V=800.0 PL=0
MOVL C01689 V=800.0 PL=0
MOVL C01690 V=800.0 PL=0
MOVL C01691 V=800.0 PL=0
MOVL C01692 V=800.0 PL=0
MOVL C01693 V=800.0 PL=0
MOVL C01694 V=800.0 PL=0
MOVL C01695 V=800.0 PL=0
MOVL C01696 V=800.0 PL=0
MOVL C01697 V=800.0 PL=0
MOVL C01698 V=800.0 PL=0
MOVL C01699 V=800.0 PL=0
MOVL C01700 V=800.0 PL=0
MOVL C01701 V=800.0 PL=0
MOVL C01702 V=800.0 PL=0
MOVL C01703 V=800.0 PL=0
MOVL C01704 V=800.0 PL=0
MOVL C01705 V=800.0 PL=0
MOVL C01706 V=800.0 PL=0
MOVL C01707 V=800.0 PL=0
MOVL C01708 V=800.0 PL=0
MOVL C01709 V=800.0 PL=0
MOVL C01710 V=800.0 PL=0
MOVL C01711 V=800.0 PL=0
MOVL C01712 V=800.0 PL=0
MOVL C01713 V=800.0 PL=0
MOVL C01714 V=800.0 PL=0
MOVL C01715 V=800.0 PL=0
MOVL C01716 V=800.0 PL=0
MOVL C01717 V=800.0 PL=0
MOVL C01718 V=800.0 PL=0
MOVL C01719 V=800.0 PL=0
MOVL C01720 V=800.0 PL=0
MOVL C01721 V=800.0 PL=0
MOVL C01722 V=800.0 PL=0
MOVL C01723 V=800.0 PL=0
MOVL C01724 V=800.0 PL=0
MOVL C01725 V=800.0 PL=0
MOVL C01726 V=800.0 PL=0
MOVL C01727 V=800.0 PL=0
MOVL C01728 V=800.0 PL=0
MOVL C01729 V=800.0 PL=0
MOVL C01730 V=800.0 PL=0
MOVL C01731 V=800.0 PL=0
MOVL C01732 V=800.0 PL=0
MOVL C01733 V=800.0 PL=0
MOVL C01734 V=800.0 PL=0
MOVL C01735 V=800.0 PL=0
MOVL C01736 V=800.0 PL=0
MOVL C01737 V=800.0 PL=0
MOVL C01738 V=800.0 PL=0
MOVL C01739 V=800.0 PL=0
MOVL C01740 V=800.0 PL=0
MOVL C01741 V=800.0 PL=0
MOVL C01742 V=800.0 PL=0
MOVL C01743 V=800.0 PL=0
MOVL C01744 V=800.0 PL=0
MOVL C01745 V=800.0 PL=0
MOVL C01746 V=800.0 PL=0
MOVL C01747 V=800.0 PL=0
MOVL C01748 V=800.0 PL=0
MOVL C01749 V=800.0 PL=0
MOVL C01750 V=800.0 PL=0
MOVL C01751 V=800.0 PL=0
MOVL C01752 V=800.0 PL=0
MOVL C01753 V=800.0 PL=0
MOVL C01754 V=800.0 PL=0
MOVL C01755 V=800.0 PL=0
MOVL C01756 V=800.0 PL=0
MOVL C01757 V=800.0 PL=0
MOVL C01758 V=800.0 PL=0
MOVL C01759 V=800.0 PL=0
MOVL C01760 V=800.0 PL=0
MOVL C01761 V=800.0 PL=0
MOVL C01762 V=800.0 PL=0
MOVL C01763 V=800.0 PL=0
MOVL C01764 V=800.0 PL=0
MOVL C01765 V=800.0 PL=0
MOVL C01766 V=800.0 PL=0
MOVL C01767 V=800.0 PL=0
MOVL C01768 V=800.0 PL=0
MOVL C01769 V=800.0 PL=0
MOVL C01770 V=800.0 PL=0
MOVL C01771 V=800.0 PL=0
MOVL C01772 V=800.0 PL=0
MOVL C01773 V=800.0 PL=0
MOVL C01774 V=800.0 PL=0
MOVL C01775 V=800.0 PL=0
MOVL C01776 V=800.0 PL=0
MOVL C01777 V=800.0 PL=0
MOVL C01778 V=800.0 PL=0
MOVL C01779 V=800.0 PL=0
MOVL C01780 V=800.0 PL=0
MOVL C01781 V=800.0 PL=0
MOVL C01782 V=800.0 PL=0
MOVL C01783 V=800.0 PL=0
MOVL C01784 V=800.0 PL=0
MOVL C01785 V=800.0 PL=0
MOVL C01786 V=800.0 PL=0
MOVL C01787 V=800.0 PL=0
MOVL C01788 V=800.0 PL=0
MOVL C01789 V=800.0 PL=0
MOVL C01790 V=800.0 PL=0
MOVL C01791 V=800.0 PL=0
MOVL C01792 V=800.0 PL=0
MOVL C01793 V=800.0 PL=0
MOVL C01794 V=800.0 PL=0
MOVL C01795 V=800.0 PL=0
MOVL C01796 V=800.0 PL=0
MOVL C01797 V=800.0 PL=0
MOVL C01798 V=800.0 PL=0
MOVL C01799 V=800.0 PL=0
MOVL C01800 V=800.0 PL=0
MOVL C01801 V=800.0 PL=0
MOVL C01802 V=800.0 PL=0
MOVL C01803 V=800.0 PL=0
MOVL C01804 V=800.0 PL=0
MOVL C01805 V=800.0 PL=0
MOVL C01806 V=800.0 PL=0
MOVL C01807 V=800.0 PL=0
MOVL C01808 V=800.0 PL=0
MOVL C01809 V=800.0 PL=0
MOVL C01810 V=800.0 PL=0
MOVL C01811 V=800.0 PL=0
MOVL C01812 V=800.0 PL=0
MOVL C01813 V=800.0 PL=0
MOVL C01814 V=800.0 PL=0
MOVL C01815 V=800.0 PL=0
MOVL C01816 V=800.0 PL=0
MOVL C01817 V=800.0 PL=0
MOVL C01818 V=800.0 PL=0
MOVL C01819 V=800.0 PL=0
MOVL C01820 V=800.0 PL=0
MOVL C01821 V=800.0 PL=0
MOVL C01822 V=800.0 PL=0
MOVL C01823 V=800.0 PL=0
MOVL C01824 V=800.0 PL=0
MOVL C01825 V=800.0 PL=0
MOVL C01826 V=800.0 PL=0
MOVL C01827 V=800.0 PL=0
MOVL C01828 V=800.0 PL=0
MOVL C01829 V=800.0 PL=0
MOVL C01830 V=800.0 PL=0
MOVL C01831 V=800.0 PL=0
MOVL C01832 V=800.0 PL=0
MOVL C01833 V=800.0 PL=0
MOVL C01834 V=800.0 PL=0
MOVL C01835 V=800.0 PL=0
MOVL C01836 V=800.0 PL=0
MOVL C01837 V=800.0 PL=0
MOVL C01838 V=800.0 PL=0
MOVL C01839 V=800.0 PL=0
MOVL C01840 V=800.0 PL=0
MOVL C01841 V=800.0 PL=0
MOVL C01842 V=800.0 PL=0
MOVL C01843 V=800.0 PL=0
MOVL C01844 V=800.0 PL=0
MOVL C01845 V=800.0 PL=0
MOVL C01846 V=800.0 PL=0
MOVL C01847 V=800.0 PL=0
MOVL C01848 V=800.0 PL=0
MOVL C01849 V=800.0 PL=0
MOVL C01850 V=800.0 PL=0
MOVL C01851 V=800.0 PL=0
MOVL C01852 V=800.0 PL=0
MOVL C01853 V=800.0 PL=0
MOVL C01854 V=800.0 PL=0
MOVL C01855 V=800.0 PL=0
MOVL C01856 V=800.0 PL=0
MOVL C01857 V=800.0 PL=0
MOVL C01858 V=800.0 PL=0
MOVL C01859 V=800.0 PL=0
MOVL C01860 V=800.0 PL=0
MOVL C01861 V=800.0 PL=0
MOVL C01862 V=800.0 PL=0
MOVL C01863 V=800.0 PL=0
MOVL C01864 V=800.0 PL=0
MOVL C01865 V=800.0 PL=0
MOVL C01866 V=800.0 PL=0
MOVL C01867 V=800.0 PL=0
MOVL C01868 V=800.0 PL=0
MOVL C01869 V=800.0 PL=0
MOVL C01870 V=800.0 PL=0
MOVL C01871 V=800.0 PL=0
MOVL C01872 V=800.0 PL=0
MOVL C01873 V=800.0 PL=0
MOVL C01874 V=800.0 PL=0
MOVL C01875 V=800.0 PL=0
MOVL C01876 V=800.0 PL=0
MOVL C01877 V=800.0 PL=0
